C01795=1066.045,135.262,-76.737,172.704,28.495,155.211
C01796=1066.039,135.013,-76.716,172.702,28.492,155.211
C01797=1066.033,134.764,-76.696,172.701,28.489,155.210
C01798=1066.028,134.516,-76.675,172.699,28.487,155.210
C01799=1066.022,134.266,-76.654,172.697,28.484,155.209
C01800=1066.016,134.017,-76.634,172.696,28.481,155.209
C01801=1066.011,133.768,-76.613,172.694,28.478,155.209
C01802=1066.004,133.518,-76.593,172.693,28.476,155.208
C01803=1065.999,133.269,-76.572,172.691,28.473,155.208
C01804=1065.993,133.020,-76.552,172.689,28.470,155.207
C01805=1065.988,132.771,-76.532,172.687,28.467,155.207
C01806=1065.982,132.522,-76.511,172.685,28.465,155.207
C01807=1065.975,132.273,-76.490,172.684,28.462,155.206
C01808=1065.970,132.024,-76.470,172.682,28.459,155.206
C01809=1065.964,131.775,-76.450,172.680,28.456,155.205
C01810=1065.958,131.526,-76.429,172.679,28.454,155.205
C01811=1065.952,131.277,-76.409,172.677,28.451,155.205
C01812=1065.946,131.028,-76.389,172.676,28.448,155.204
C01813=1065.940,130.779,-76.369,172.674,28.445,155.204
C01814=1065.934,130.529,-76.348,172.673,28.443,155.203
C01815=1065.928,130.280,-76.328,172.671,28.440,155.203
C01816=1065.922,130.032,-76.308,172.669,28.438,155.203
C01817=1065.917,129.783,-76.288,172.667,28.435,155.202
C01818=1065.911,129.533,-76.267,172.665,28.432,155.202
C01819=1065.905,129.284,-76.247,172.664,28.429,155.201
C01820=1065.899,129.035,-76.228,172.662,28.426,155.201
C01821=1065.894,128.786,-76.208,172.660,28.424,155.201
C01822=1065.887,128.536,-76.187,172.659,28.421,155.200
C01823=1065.881,128.287,-76.167,172.657,28.418,155.200
C01824=1065.876,128.038,-76.147,172.656,28.416,155.200
C01825=1065.870,127.789,-76.127,172.654,28.413,155.199
C01826=1065.863,127.540,-76.106,172.652,28.410,155.199
C01827=1065.857,127.291,-76.086,172.651,28.408,155.198
C01828=1065.851,127.007,-76.064,172.648,28.404,155.198
C01829=1065.845,126.724,-76.041,172.647,28.401,155.197
C01830=1065.837,126.440,-76.018,172.645,28.398,155.197
C01831=1065.831,126.157,-75.995,172.643,28.395,155.197
C01832=1065.826,125.907,-75.975,172.641,28.392,155.196
C01833=1065.820,125.658,-75.955,172.640,28.390,155.196
C01834=1065.814,125.409,-75.935,172.638,28.387,155.195
C01835=1065.807,125.160,-75.915,172.636,28.384,155.195
C01836=1065.802,124.911,-75.894,172.635,28.381,155.195
C01837=1065.796,124.662,-75.874,172.633,28.379,155.194
C01838=1065.790,124.412,-75.855,172.632,28.376,155.194
C01839=1065.784,124.164,-75.835,172.630,28.373,155.193
C01840=1065.779,123.914,-75.814,172.628,28.370,155.193
C01841=1065.772,123.665,-75.794,172.627,28.368,155.193
C01842=1065.767,123.416,-75.775,172.625,28.365,155.192
C01843=1065.761,123.167,-75.755,172.624,28.363,155.192
C01844=1065.755,122.918,-75.735,172.622,28.360,155.191
C01845=1065.749,122.669,-75.714,172.620,28.357,155.191
C01846=1065.744,122.419,-75.695,172.619,28.354,155.191
C01847=1065.738,122.171,-75.675,172.617,28.352,155.190
C01848=1065.732,121.922,-75.655,172.616,28.349,155.190
C01849=1065.727,121.672,-75.635,172.614,28.346,155.189
C01850=1065.721,121.423,-75.615,172.612,28.343,155.189
C01851=1065.714,121.174,-75.595,172.610,28.340,155.189
C01852=1065.708,120.924,-75.576,172.608,28.337,155.188
C01853=1065.702,120.675,-75.556,172.607,28.335,155.188
C01854=1065.697,120.426,-75.535,172.605,28.332,155.187
C01855=1065.692,120.177,-75.516,172.604,28.329,155.187
C01856=1065.686,119.928,-75.496,172.602,28.326,155.187
C01857=1065.680,119.679,-75.476,172.601,28.324,155.186
C01858=1065.674,119.430,-75.457,172.599,28.321,155.186
C01859=1065.669,119.181,-75.436,172.597,28.318,155.185
C01860=1065.663,118.931,-75.417,172.596,28.315,155.185
C01861=1065.657,118.682,-75.397,172.594,28.313,155.185
C01862=1065.651,118.434,-75.377,172.593,28.310,155.184
C01863=1065.645,118.184,-75.358,172.591,28.307,155.184
C01864=1065.639,117.935,-75.338,172.589,28.304,155.183
C01865=1065.634,117.686,-75.318,172.588,28.302,155.183
C01866=1065.628,117.437,-75.298,172.586,28.299,155.183
C01867=1065.623,117.187,-75.279,172.585,28.296,155.182
C01868=1065.617,116.939,-75.259,172.583,28.293,155.182
C01869=1065.611,116.689,-75.240,172.582,28.291,155.181
C01870=1065.605,116.440,-75.220,172.580,28.288,155.181
C01871=1065.600,116.191,-75.200,172.578,28.285,155.181
C01872=1065.594,115.942,-75.180,172.577,28.282,155.180
C01873=1065.588,115.692,-75.161,172.575,28.280,155.180
C01874=1065.582,115.444,-75.141,172.574,28.277,155.179
C01875=1065.577,115.194,-75.122,172.572,28.274,155.179
C01876=1065.571,114.945,-75.102,172.571,28.271,155.178
C01877=1065.565,114.696,-75.082,172.569,28.268,155.178
C01878=1065.560,114.447,-75.062,172.568,28.265,155.178
C01879=1065.554,114.197,-75.043,172.566,28.262,155.177
C01880=1065.548,113.948,-75.023,172.564,28.260,155.177
C01881=1065.542,113.699,-75.003,172.563,28.257,155.176
C01882=1065.537,113.450,-74.984,172.561,28.255,155.176
C01883=1065.530,113.201,-74.965,172.560,28.252,155.176
C01884=1065.524,112.952,-74.946,172.558,28.249,155.175
C01885=1065.519,112.702,-74.926,172.556,28.246,155.175
C01886=1065.513,112.453,-74.906,172.555,28.244,155.174
C01887=1065.507,112.204,-74.887,172.553,28.241,155.174
C01888=1065.501,111.955,-74.868,172.552,28.238,155.174
C01889=1065.495,111.706,-74.848,172.550,28.235,155.173
C01890=1065.489,111.456,-74.829,172.549,28.232,155.173
C01891=1065.484,111.207,-74.809,172.547,28.230,155.172
C01892=1065.477,110.923,-74.787,172.545,28.227,155.172
C01893=1065.470,110.640,-74.765,172.543,28.223,155.172
C01894=1065.463,110.356,-74.743,172.541,28.221,155.171
C01895=1065.457,110.072,-74.721,172.540,28.217,155.171
C01896=1065.450,109.823,-74.702,172.538,28.215,155.170
C01897=1065.445,109.574,-74.683,172.537,28.212,155.170
C01898=1065.439,109.325,-74.664,172.535,28.210,155.170
C01899=1065.433,109.075,-74.644,172.534,28.207,155.169
C01900=1065.427,108.826,-74.624,172.532,28.204,155.169
C01901=1065.421,108.577,-74.606,172.530,28.201,155.168
C01902=1065.415,108.328,-74.586,172.529,28.198,155.168
C01903=1065.410,108.078,-74.567,172.527,28.196,155.168
C01904=1065.404,107.830,-74.548,172.526,28.193,155.167
C01905=1065.398,107.581,-74.529,172.524,28.190,155.167
C01906=1065.392,107.332,-74.510,172.523,28.187,155.166
C01907=1065.386,107.082,-74.490,172.521,28.185,155.166
C01908=1065.381,106.833,-74.471,172.519,28.182,155.166
C01909=1065.374,106.584,-74.453,172.518,28.180,155.165
C01910=1065.369,106.334,-74.433,172.516,28.177,155.165
C01911=1065.363,106.085,-74.414,172.515,28.174,155.164
C01912=1065.357,105.836,-74.394,172.513,28.171,155.164
C01913=1065.350,105.587,-74.375,172.512,28.169,155.164
C01914=1065.345,105.338,-74.357,172.510,28.166,155.163
C01915=1065.340,105.089,-74.337,172.508,28.163,155.163
C01916=1065.334,104.839,-74.318,172.507,28.160,155.162
C01917=1065.328,104.590,-74.299,172.505,28.157,155.162
C01918=1065.322,104.341,-74.280,172.504,28.155,155.162
C01919=1065.316,104.091,-74.261,172.502,28.152,155.161
C01920=1065.310,103.842,-74.242,172.501,28.149,155.161
C01921=1065.305,103.593,-74.223,172.499,28.146,155.160
C01922=1065.299,103.344,-74.204,172.498,28.144,155.160
C01923=1065.293,103.095,-74.185,172.497,28.141,155.160
C01924=1065.287,102.845,-74.166,172.495,28.138,155.159
C01925=1065.281,102.596,-74.147,172.494,28.136,155.159
C01926=1065.275,102.347,-74.128,172.492,28.133,155.158
C01927=1065.270,102.098,-74.110,172.491,28.130,155.158
C01928=1065.264,101.849,-74.090,172.489,28.127,155.158
C01929=1065.258,101.599,-74.071,172.488,28.124,155.157
C01930=1065.253,101.350,-74.052,172.486,28.122,155.157
C01931=1065.246,101.101,-74.033,172.484,28.119,155.156
C01932=1065.241,100.852,-74.014,172.483,28.116,155.156
C01933=1065.235,100.603,-73.996,172.481,28.114,155.156
C01934=1065.229,100.353,-73.976,172.480,28.111,155.155
C01935=1065.223,100.104,-73.958,172.478,28.108,155.155
C01936=1065.217,99.855,-73.939,172.477,28.106,155.154
C01937=1065.210,99.606,-73.920,172.475,28.103,155.154
C01938=1065.205,99.356,-73.901,172.473,28.100,155.154
C01939=1065.199,99.108,-73.882,172.472,28.097,155.153
C01940=1065.193,98.859,-73.863,172.470,28.094,155.153
C01941=1065.187,98.609,-73.845,172.469,28.092,155.153
C01942=1065.181,98.359,-73.826,172.467,28.089,155.152
C01943=1065.175,98.110,-73.807,172.466,28.087,155.152
C01944=1065.170,97.862,-73.788,172.464,28.084,155.151
C01945=1065.163,97.612,-73.770,172.462,28.081,155.151
C01946=1065.158,97.363,-73.751,172.461,28.078,155.151
C01947=1065.151,97.114,-73.732,172.460,28.076,155.150
C01948=1065.146,96.864,-73.713,172.459,28.073,155.150
C01949=1065.140,96.615,-73.695,172.457,28.070,155.149
C01950=1065.134,96.366,-73.676,172.456,28.067,155.149
C01951=1065.128,96.117,-73.657,172.454,28.065,155.149
C01952=1065.122,95.867,-73.639,172.452,28.062,155.148
C01953=1065.117,95.618,-73.620,172.451,28.060,155.148
C01954=1065.110,95.369,-73.602,172.449,28.057,155.147
C01955=1065.105,95.120,-73.582,172.448,28.054,155.147
C01956=1065.098,94.836,-73.561,172.446,28.051,155.147
C01957=1065.091,94.553,-73.541,172.445,28.048,155.146
C01958=1065.085,94.268,-73.519,172.442,28.044,155.146
C01959=1065.078,93.985,-73.497,172.441,28.042,155.145
C01960=1065.072,93.736,-73.480,172.439,28.039,155.145
C01961=1065.067,93.486,-73.461,172.438,28.036,155.144
C01962=1065.060,93.237,-73.442,172.436,28.033,155.144
C01963=1065.055,92.988,-73.424,172.435,28.030,155.144
C01964=1065.049,92.739,-73.405,172.433,28.028,155.143
C01965=1065.043,92.490,-73.387,172.431,28.025,155.143
C01966=1065.037,92.240,-73.368,172.431,28.022,155.142
C01967=1065.031,91.991,-73.350,172.429,28.020,155.142
C01968=1065.026,91.742,-73.330,172.428,28.017,155.142
C01969=1065.020,91.492,-73.313,172.426,28.014,155.141
C01970=1065.014,91.244,-73.294,172.425,28.011,155.141
C01971=1065.008,90.994,-73.275,172.423,28.009,155.141
C01972=1065.002,90.745,-73.257,172.421,28.006,155.140
C01973=1064.996,90.496,-73.239,172.420,28.003,155.140
C01974=1064.991,90.246,-73.220,172.418,28.001,155.139
C01975=1064.984,89.997,-73.202,172.417,27.998,155.139
C01976=1064.979,89.748,-73.184,172.415,27.995,155.139
C01977=1064.972,89.499,-73.165,172.414,27.992,155.138
C01978=1064.966,89.250,-73.147,172.412,27.990,155.138
C01979=1064.961,89.000,-73.128,172.410,27.987,155.137
C01980=1064.955,88.751,-73.110,172.409,27.985,155.137
C01981=1064.949,88.501,-73.092,172.408,27.982,155.137
C01982=1064.942,88.252,-73.073,172.407,27.979,155.136
C01983=1064.937,88.003,-73.056,172.405,27.976,155.136
C01984=1064.931,87.754,-73.037,172.404,27.974,155.135
C01985=1064.925,87.504,-73.019,172.402,27.971,155.135
C01986=1064.919,87.256,-73.000,172.401,27.969,155.135
C01987=1064.913,87.006,-72.982,172.399,27.966,155.134
C01988=1064.906,86.757,-72.964,172.397,27.963,155.134
C01989=1064.901,86.508,-72.946,172.396,27.960,155.134
C01990=1064.896,86.258,-72.928,172.394,27.957,155.133
C01991=1064.889,86.009,-72.909,172.393,27.955,155.133
C01992=1064.884,85.760,-72.891,172.391,27.952,155.132
C01993=1064.877,85.510,-72.873,172.390,27.949,155.132
C01994=1064.871,85.261,-72.855,172.388,27.947,155.132
C01995=1064.865,85.012,-72.837,172.387,27.944,155.131
C01996=1064.859,84.763,-72.819,172.386,27.942,155.131
C01997=1064.854,84.513,-72.800,172.384,27.939,155.130
C01998=1064.848,84.264,-72.782,172.383,27.936,155.130
C01999=1064.842,84.014,-72.764,172.381,27.933,155.130
C02000=1064.836,83.766,-72.746,172.380,27.930,155.129
C02001=1064.830,83.516,-72.728,172.378,27.928,155.129
C02002=1064.824,83.267,-72.710,172.377,27.925,155.128
C02003=1064.818,83.018,-72.691,172.375,27.922,155.128
C02004=1064.812,82.768,-72.674,172.373,27.920,155.128
C02005=1064.807,82.519,-72.655,172.372,27.917,155.127
C02006=1064.801,82.270,-72.637,172.370,27.914,155.127
C02007=1064.795,82.021,-72.619,172.370,27.912,155.127
C02008=1064.789,81.771,-72.601,172.368,27.909,155.126
C02009=1064.783,81.522,-72.584,172.367,27.906,155.126
C02010=1064.777,81.273,-72.565,172.365,27.903,155.125
C02011=1064.771,81.024,-72.547,172.364,27.900,155.125
C02012=1064.765,80.774,-72.530,172.362,27.898,155.125
C02013=1064.760,80.526,-72.511,172.361,27.895,155.124
C02014=1064.754,80.276,-72.493,172.359,27.892,155.124
C02015=1064.748,80.026,-72.475,172.357,27.889,155.123
C02016=1064.743,79.777,-72.457,172.356,27.887,155.123
C02017=1064.736,79.528,-72.439,172.354,27.884,155.123
C02018=1064.731,79.279,-72.421,172.354,27.882,155.122
C02019=1064.724,79.029,-72.403,172.352,27.879,155.122
C02020=1064.718,78.746,-72.382,172.350,27.875,155.121
C02021=1064.711,78.462,-72.363,172.348,27.873,155.121
C02022=1064.704,78.178,-72.342,172.347,27.869,155.120
C02023=1064.698,77.894,-72.322,172.345,27.866,155.120
C02024=1064.692,77.645,-72.303,172.344,27.864,155.120
C02025=1064.686,77.396,-72.286,172.342,27.861,155.119
C02026=1064.680,77.146,-72.268,172.341,27.858,155.119
C02027=1064.674,76.898,-72.251,172.339,27.855,155.118
C02028=1064.668,76.648,-72.233,172.338,27.853,155.118
C02029=1064.662,76.399,-72.216,172.336,27.850,155.118
C02030=1064.656,76.149,-72.198,172.335,27.848,155.117
C02031=1064.650,75.901,-72.179,172.334,27.845,155.117
C02032=1064.644,75.651,-72.161,172.332,27.842,155.117
C02033=1064.639,75.402,-72.144,172.331,27.839,155.116
C02034=1064.633,75.152,-72.126,172.329,27.836,155.116
C02035=1064.626,74.903,-72.109,172.328,27.834,155.115
C02036=1064.620,74.654,-72.091,172.326,27.831,155.115
C02037=1064.615,74.405,-72.073,172.325,27.829,155.115
C02038=1064.609,74.155,-72.055,172.323,27.826,155.114
C02039=1064.603,73.906,-72.038,172.321,27.823,155.114
C02040=1064.597,73.656,-72.020,172.321,27.820,155.113
C02041=1064.591,73.407,-72.002,172.319,27.818,155.113
C02042=1064.585,73.158,-71.985,172.318,27.815,155.113
C02043=1064.579,72.909,-71.967,172.316,27.813,155.112
C02044=1064.573,72.659,-71.950,172.315,27.810,155.112
C02045=1064.567,72.410,-71.932,172.313,27.807,155.112
C02046=1064.561,72.160,-71.914,172.312,27.804,155.111
C02047=1064.556,71.911,-71.896,172.310,27.801,155.111
C02048=1064.549,71.662,-71.880,172.309,27.799,155.110
C02049=1064.543,71.413,-71.862,172.307,27.796,155.110
C02050=1064.538,71.164,-71.844,172.305,27.794,155.110
C02051=1064.532,70.914,-71.826,172.305,27.791,155.109
C02052=1064.526,70.665,-71.809,172.303,27.788,155.109
C02053=1064.519,70.415,-71.791,172.302,27.785,155.108
C02054=1064.514,70.166,-71.774,172.300,27.783,155.108
C02055=1064.508,69.917,-71.756,172.299,27.780,155.108
C02056=1064.502,69.667,-71.739,172.297,27.777,155.107
C02057=1064.496,69.418,-71.722,172.296,27.774,155.107
C02058=1064.490,69.168,-71.704,172.294,27.772,155.107
C02059=1064.485,68.919,-71.686,172.292,27.769,155.106
C02060=1064.478,68.670,-71.669,172.292,27.767,155.106
C02061=1064.472,68.421,-71.651,172.290,27.764,155.105
C02062=1064.467,68.172,-71.634,172.289,27.761,155.105
C02063=1064.460,67.922,-71.617,172.287,27.758,155.105
C02064=1064.455,67.673,-71.600,172.286,27.756,155.104
C02065=1064.449,67.423,-71.582,172.284,27.753,155.104
C02066=1064.442,67.174,-71.565,172.283,27.750,155.104
C02067=1064.437,66.925,-71.547,172.281,27.748,155.103
C02068=1064.431,66.676,-71.529,172.280,27.745,155.103
C02069=1064.425,66.426,-71.513,172.278,27.742,155.102
C02070=1064.419,66.176,-71.495,172.277,27.740,155.102
C02071=1064.413,65.927,-71.478,172.276,27.737,155.102
C02072=1064.407,65.679,-71.461,172.274,27.734,155.101
C02073=1064.401,65.428,-71.443,172.273,27.732,155.101
C02074=1064.395,65.180,-71.426,172.271,27.729,155.100
C02075=1064.389,64.931,-71.409,172.270,27.726,155.100
C02076=1064.383,64.681,-71.391,172.268,27.723,155.100
C02077=1064.377,64.431,-71.375,172.267,27.721,155.099
C02078=1064.371,64.182,-71.357,172.265,27.718,155.099
C02079=1064.365,63.933,-71.340,172.265,27.716,155.099
C02080=1064.360,63.683,-71.323,172.263,27.713,155.098
C02081=1064.353,63.434,-71.306,172.261,27.711,155.098
C02082=1064.346,63.185,-71.289,172.260,27.708,155.097
C02083=1064.340,62.935,-71.271,172.258,27.705,155.097
C02084=1064.334,62.651,-71.252,172.257,27.702,155.097
C02085=1064.327,62.368,-71.233,172.255,27.699,155.096
C02086=1064.320,62.084,-71.213,172.253,27.696,155.096
C02087=1064.313,61.800,-71.194,172.251,27.693,155.095
C02088=1064.306,61.551,-71.177,172.250,27.691,155.095
C02089=1064.301,61.302,-71.159,172.248,27.688,155.095
C02090=1064.294,61.052,-71.142,172.248,27.685,155.094
C02091=1064.289,60.803,-71.125,172.246,27.682,155.094
C02092=1064.282,60.553,-71.108,172.245,27.680,155.094
C02093=1064.276,60.304,-71.091,172.243,27.677,155.093
C02094=1064.271,60.055,-71.074,172.242,27.675,155.093
C02095=1064.264,59.805,-71.057,172.240,27.672,155.092
C02096=1064.258,59.556,-71.040,172.238,27.670,155.092
C02097=1064.253,59.307,-71.023,172.237,27.667,155.092
C02098=1064.246,59.057,-71.006,172.235,27.664,155.091
C02099=1064.240,58.808,-70.990,172.235,27.661,155.091
C02100=1064.234,58.559,-70.972,172.233,27.659,155.091
C02101=1064.228,58.310,-70.956,172.232,27.656,155.090
C02102=1064.222,58.060,-70.938,172.230,27.653,155.090
C02103=1064.216,57.810,-70.922,172.229,27.651,155.089
C02104=1064.210,57.562,-70.905,172.227,27.648,155.089
C02105=1064.204,57.311,-70.887,172.225,27.646,155.089
C02106=1064.198,57.063,-70.871,172.224,27.643,155.088
C02107=1064.192,56.813,-70.854,172.222,27.640,155.088
C02108=1064.186,56.564,-70.837,172.222,27.637,155.088
C02109=1064.180,56.314,-70.820,172.220,27.635,155.087
C02110=1064.174,56.065,-70.803,172.219,27.632,155.087
C02111=1064.168,55.816,-70.786,172.217,27.630,155.087
C02112=1064.162,55.566,-70.769,172.216,27.627,155.086
C02113=1064.156,55.317,-70.753,172.214,27.624,155.086
C02114=1064.150,55.068,-70.736,172.213,27.622,155.085
C02115=1064.144,54.819,-70.719,172.211,27.619,155.085
C02116=1064.138,54.569,-70.703,172.210,27.616,155.085
C02117=1064.131,54.320,-70.685,172.209,27.613,155.084
C02118=1064.126,54.070,-70.668,172.207,27.611,155.084
C02119=1064.120,53.821,-70.652,172.206,27.608,155.084
C02120=1064.114,53.572,-70.635,172.204,27.606,155.083
C02121=1064.108,53.322,-70.618,172.203,27.603,155.083
C02122=1064.102,53.072,-70.602,172.201,27.601,155.082
C02123=1064.096,52.824,-70.585,172.200,27.598,155.082
C02124=1064.091,52.574,-70.568,172.198,27.595,155.082
C02125=1064.085,52.325,-70.552,172.197,27.592,155.081
C02126=1064.078,52.075,-70.534,172.196,27.590,155.081
C02127=1064.072,51.826,-70.518,172.195,27.587,155.081
C02128=1064.067,51.576,-70.501,172.193,27.584,155.080
C02129=1064.060,51.327,-70.484,172.192,27.582,155.080
C02130=1064.054,51.078,-70.468,172.190,27.579,155.079
C02131=1064.049,50.828,-70.451,172.188,27.576,155.079
C02132=1064.042,50.579,-70.434,172.187,27.574,155.079
C02133=1064.036,50.330,-70.417,172.185,27.571,155.078
C02134=1064.030,50.080,-70.401,172.185,27.568,155.078
C02135=1064.025,49.831,-70.384,172.183,27.566,155.078
C02136=1064.019,49.582,-70.367,172.182,27.563,155.077
C02137=1064.013,49.333,-70.351,172.180,27.560,155.077
C02138=1064.007,49.083,-70.335,172.179,27.558,155.076
C02139=1064.001,48.833,-70.318,172.177,27.555,155.076
C02140=1063.995,48.584,-70.301,172.176,27.552,155.076
C02141=1063.989,48.335,-70.284,172.174,27.549,155.075
C02142=1063.983,48.085,-70.268,172.173,27.546,155.075
C02143=1063.978,47.836,-70.251,172.172,27.544,155.075
C02144=1063.972,47.586,-70.235,172.170,27.542,155.074
C02145=1063.966,47.337,-70.219,172.169,27.539,155.074
C02146=1063.960,47.088,-70.202,172.167,27.536,155.073
C02147=1063.955,46.839,-70.185,172.166,27.533,155.073
C02148=1063.948,46.555,-70.166,172.164,27.530,155.073
C02149=1063.940,46.270,-70.148,172.163,27.527,155.072
C02150=1063.933,45.986,-70.129,172.162,27.524,155.072
C02151=1063.927,45.702,-70.110,172.160,27.521,155.071
C02152=1063.922,45.453,-70.093,172.159,27.518,155.071
C02153=1063.916,45.203,-70.077,172.157,27.516,155.070
C02154=1063.910,44.954,-70.061,172.156,27.513,155.070
C02155=1063.904,44.704,-70.044,172.154,27.510,155.070
C02156=1063.898,44.455,-70.028,172.152,27.508,155.069
C02157=1063.893,44.205,-70.011,172.151,27.505,155.069
C02158=1063.886,43.957,-69.994,172.149,27.502,155.069
C02159=1063.880,43.707,-69.978,172.148,27.499,155.068
C02160=1063.874,43.458,-69.962,172.147,27.497,155.068
C02161=1063.869,43.209,-69.946,172.146,27.494,155.068
C02162=1063.863,42.959,-69.929,172.144,27.492,155.067
C02163=1063.856,42.709,-69.913,172.143,27.489,155.067
C02164=1063.850,42.460,-69.896,172.141,27.486,155.066
C02165=1063.844,42.211,-69.880,172.140,27.484,155.066
C02166=1063.838,41.961,-69.864,172.138,27.481,155.066
C02167=1063.832,41.712,-69.848,172.137,27.478,155.065
C02168=1063.826,41.463,-69.831,172.136,27.476,155.065
C02169=1063.820,41.213,-69.815,172.134,27.473,155.065
C02170=1063.814,40.964,-69.799,172.133,27.470,155.064
C02171=1063.808,40.715,-69.783,172.131,27.468,155.064
C02172=1063.802,40.465,-69.766,172.130,27.465,155.064
C02173=1063.797,40.215,-69.751,172.128,27.462,155.063
C02174=1063.791,39.966,-69.735,172.127,27.460,155.063
C02175=1063.785,39.717,-69.718,172.125,27.457,155.062
C02176=1063.779,39.467,-69.702,172.124,27.455,155.062
C02177=1063.773,39.218,-69.686,172.123,27.452,155.062
C02178=1063.767,38.968,-69.670,172.122,27.449,155.061
C02179=1063.761,38.719,-69.653,172.120,27.447,155.061
C02180=1063.755,38.470,-69.637,172.119,27.444,155.061
C02181=1063.749,38.220,-69.621,172.117,27.441,155.060
C02182=1063.743,37.971,-69.605,172.116,27.438,155.060
C02183=1063.738,37.721,-69.589,172.114,27.436,155.060
C02184=1063.731,37.472,-69.573,172.113,27.433,155.059
C02185=1063.725,37.223,-69.557,172.111,27.431,155.059
C02186=1063.719,36.973,-69.541,172.110,27.429,155.058
C02187=1063.713,36.724,-69.525,172.109,27.426,155.058
C02188=1063.707,36.475,-69.508,172.107,27.423,155.058
C02189=1063.701,36.225,-69.493,172.106,27.421,155.057
C02190=1063.695,35.976,-69.477,172.104,27.418,155.057
C02191=1063.689,35.726,-69.461,172.103,27.416,155.057
C02192=1063.683,35.477,-69.445,172.101,27.413,155.056
C02193=1063.677,35.228,-69.428,172.100,27.410,155.056
C02194=1063.671,34.978,-69.413,172.098,27.408,155.056
C02195=1063.665,34.729,-69.397,172.098,27.405,155.055
C02196=1063.659,34.479,-69.381,172.096,27.402,155.055
C02197=1063.653,34.230,-69.365,172.094,27.400,155.055
C02198=1063.646,33.980,-69.350,172.093,27.397,155.054
C02199=1063.640,33.731,-69.333,172.091,27.394,155.054
C02200=1063.634,33.482,-69.317,172.090,27.392,155.053
C02201=1063.629,33.232,-69.302,172.088,27.389,155.053
C02202=1063.622,32.983,-69.286,172.087,27.386,155.053
C02203=1063.616,32.733,-69.270,172.086,27.384,155.052
C02204=1063.610,32.484,-69.253,172.085,27.382,155.052
C02205=1063.605,32.234,-69.238,172.083,27.379,155.052
C02206=1063.598,31.985,-69.222,172.082,27.376,155.051
C02207=1063.592,31.736,-69.206,172.080,27.374,155.051
C02208=1063.586,31.486,-69.190,172.079,27.371,155.051
C02209=1063.580,31.236,-69.174,172.077,27.368,155.050
C02210=1063.574,30.987,-69.158,172.076,27.366,155.050
C02211=1063.569,30.738,-69.143,172.074,27.363,155.050
C02212=1063.561,30.454,-69.125,172.073,27.360,155.049
C02213=1063.555,30.170,-69.107,172.071,27.357,155.049
C02214=1063.548,29.885,-69.089,172.070,27.354,155.048
C02215=1063.541,29.601,-69.071,172.068,27.351,155.048
C02216=1063.535,29.352,-69.055,172.067,27.349,155.048
C02217=1063.529,29.102,-69.040,172.065,27.346,155.047
C02218=1063.523,28.853,-69.023,172.064,27.344,155.047
C02219=1063.517,28.603,-69.008,172.062,27.341,155.046
C02220=1063.511,28.354,-68.992,172.061,27.338,155.046
C02221=1063.506,28.105,-68.977,172.059,27.336,155.046
C02222=1063.499,27.855,-68.961,172.058,27.334,155.046
C02223=1063.493,27.605,-68.946,172.057,27.331,155.045
C02224=1063.487,27.356,-68.930,172.055,27.328,155.045
C02225=1063.481,27.106,-68.914,172.054,27.326,155.044
C02226=1063.474,26.857,-68.899,172.052,27.323,155.044
C02227=1063.469,26.607,-68.883,172.051,27.321,155.044
C02228=1063.463,26.358,-68.867,172.049,27.318,155.043
C02229=1063.456,26.108,-68.852,172.048,27.315,155.043
C02230=1063.451,25.860,-68.836,172.046,27.313,155.043
C02231=1063.445,25.610,-68.821,172.046,27.310,155.042
C02232=1063.439,25.361,-68.805,172.044,27.308,155.042
C02233=1063.432,25.111,-68.790,172.043,27.305,155.042
C02234=1063.426,24.862,-68.774,172.041,27.303,155.041
C02235=1063.420,24.612,-68.759,172.039,27.300,155.041
C02236=1063.414,24.363,-68.743,172.038,27.298,155.041
C02237=1063.408,24.114,-68.728,172.036,27.295,155.040
C02238=1063.403,23.864,-68.712,172.035,27.292,155.040
C02239=1063.396,23.615,-68.697,172.033,27.290,155.040
C02240=1063.390,23.365,-68.681,172.032,27.287,155.039
C02241=1063.384,23.116,-68.666,172.031,27.285,155.039
C02242=1063.378,22.866,-68.650,172.030,27.282,155.039
C02243=1063.372,22.617,-68.635,172.028,27.280,155.038
C02244=1063.366,22.368,-68.619,172.027,27.277,155.038
C02245=1063.360,22.118,-68.604,172.025,27.274,155.037
C02246=1063.354,21.868,-68.589,172.024,27.272,155.037
C02247=1063.347,21.619,-68.573,172.022,27.269,155.037
C02248=1063.342,21.370,-68.558,172.021,27.267,155.037
C02249=1063.336,21.120,-68.543,172.019,27.264,155.036
C02250=1063.330,20.871,-68.527,172.018,27.262,155.036
C02251=1063.324,20.621,-68.512,172.017,27.259,155.035
C02252=1063.318,20.371,-68.496,172.015,27.257,155.035
C02253=1063.312,20.123,-68.481,172.014,27.254,155.035
C02254=1063.306,19.873,-68.466,172.012,27.252,155.035
C02255=1063.300,19.623,-68.450,172.011,27.249,155.034
C02256=1063.293,19.374,-68.435,172.009,27.246,155.034
C02257=1063.287,19.124,-68.420,172.008,27.244,155.033
C02258=1063.282,18.875,-68.405,172.006,27.241,155.033
C02259=1063.275,18.625,-68.390,172.005,27.238,155.033
C02260=1063.270,18.376,-68.373,172.004,27.236,155.033
C02261=1063.263,18.126,-68.358,172.003,27.234,155.032
C02262=1063.257,17.877,-68.344,172.001,27.231,155.032
C02263=1063.252,17.628,-68.328,171.999,27.229,155.031
C02264=1063.245,17.378,-68.313,171.998,27.226,155.031
C02265=1063.239,17.129,-68.298,171.996,27.223,155.031
C02266=1063.234,16.880,-68.283,171.995,27.221,155.031
C02267=1063.227,16.630,-68.268,171.993,27.218,155.030
C02268=1063.221,16.380,-68.253,171.992,27.216,155.030
C02269=1063.215,16.130,-68.237,171.990,27.213,155.029
C02270=1063.209,15.881,-68.223,171.990,27.211,155.029
C02271=1063.203,15.632,-68.207,171.988,27.208,155.029
C02272=1063.197,15.382,-68.191,171.987,27.206,155.028
C02273=1063.191,15.133,-68.176,171.985,27.203,155.028
C02274=1063.185,14.884,-68.162,171.984,27.201,155.028
C02275=1063.179,14.634,-68.146,171.982,27.198,155.027
C02276=1063.172,14.351,-68.129,171.981,27.195,155.027
C02277=1063.165,14.069,-68.113,171.979,27.192,155.027
C02278=1063.158,13.786,-68.095,171.978,27.190,155.026
C02279=1063.151,13.503,-68.078,171.975,27.187,155.026
C02280=1063.145,13.254,-68.063,171.974,27.184,155.026
C02281=1063.139,13.004,-68.048,171.973,27.182,155.025
C02282=1063.132,12.754,-68.033,171.972,27.179,155.025
C02283=1063.126,12.505,-68.018,171.970,27.177,155.025
C02284=1063.120,12.256,-68.004,171.968,27.175,155.024
C02285=1063.114,12.006,-67.989,171.967,27.172,155.024
C02286=1063.108,11.757,-67.974,171.965,27.170,155.024
C02287=1063.103,11.507,-67.959,171.964,27.167,155.023
C02288=1063.096,11.258,-67.944,171.962,27.165,155.023
C02289=1063.090,11.008,-67.929,171.961,27.162,155.023
C02290=1063.083,10.758,-67.914,171.959,27.159,155.022
C02291=1063.078,10.509,-67.899,171.958,27.157,155.022
C02292=1063.071,10.260,-67.884,171.956,27.155,155.022
C02293=1063.065,10.010,-67.869,171.956,27.152,155.021
C02294=1063.059,9.761,-67.855,171.954,27.150,155.021
C02295=1063.053,9.511,-67.840,171.952,27.148,155.021
C02296=1063.046,9.262,-67.825,171.951,27.145,155.021
C02297=1063.040,9.013,-67.810,171.949,27.143,155.020
C02298=1063.035,8.763,-67.795,171.948,27.140,155.020
C02299=1063.028,8.513,-67.780,171.946,27.137,155.020
C02300=1063.023,8.264,-67.766,171.945,27.135,155.019
C02301=1063.017,8.014,-67.751,171.943,27.132,155.019
C02302=1063.010,7.764,-67.736,171.942,27.130,155.019
C02303=1063.004,7.515,-67.722,171.940,27.128,155.018
C02304=1062.998,7.266,-67.707,171.940,27.125,155.018
C02305=1062.992,7.017,-67.692,171.938,27.123,155.018
C02306=1062.986,6.767,-67.677,171.936,27.121,155.017
C02307=1062.980,6.517,-67.662,171.935,27.118,155.017
C02308=1062.974,6.268,-67.648,171.933,27.115,155.017
C02309=1062.968,6.018,-67.633,171.932,27.113,155.017
C02310=1062.961,5.769,-67.618,171.930,27.110,155.016
C02311=1062.955,5.520,-67.604,171.929,27.108,155.016
C02312=1062.949,5.270,-67.589,171.927,27.105,155.015
C02313=1062.943,5.021,-67.574,171.926,27.103,155.015
C02314=1062.937,4.771,-67.560,171.924,27.101,155.015
C02315=1062.931,4.522,-67.545,171.923,27.098,155.015
C02316=1062.925,4.272,-67.531,171.921,27.096,155.014
C02317=1062.919,4.022,-67.515,171.920,27.094,155.014
C02318=1062.914,3.773,-67.500,171.919,27.091,155.014
C02319=1062.908,3.523,-67.486,171.917,27.088,155.013
C02320=1062.902,3.274,-67.472,171.916,27.086,155.013
C02321=1062.895,3.024,-67.457,171.914,27.083,155.013
C02322=1062.890,2.775,-67.442,171.913,27.081,155.012
C02323=1062.884,2.525,-67.428,171.911,27.079,155.012
C02324=1062.877,2.275,-67.413,171.910,27.076,155.012
C02325=1062.871,2.026,-67.398,171.908,27.074,155.011
C02326=1062.865,1.777,-67.383,171.907,27.071,155.011
C02327=1062.860,1.527,-67.370,171.905,27.068,155.011
C02328=1062.853,1.278,-67.355,171.904,27.066,155.011
C02329=1062.847,1.029,-67.340,171.903,27.064,155.010
C02330=1062.841,0.778,-67.326,171.902,27.061,155.010
C02331=1062.835,0.529,-67.311,171.900,27.059,155.010
C02332=1062.829,0.280,-67.296,171.899,27.056,155.009
C02333=1062.824,0.030,-67.282,171.897,27.054,155.009
C02334=1062.817,-0.220,-67.267,171.895,27.052,155.009
C02335=1062.811,-0.469,-67.253,171.894,27.049,155.008
C02336=1062.805,-0.719,-67.239,171.892,27.046,155.008
C02337=1062.800,-0.968,-67.224,171.891,27.044,155.008
C02338=1062.793,-1.217,-67.209,171.889,27.041,155.007
C02339=1062.787,-1.467,-67.196,171.888,27.039,155.007
C02340=1062.781,-1.747,-67.179,171.886,27.036,155.007
C02341=1062.774,-2.029,-67.163,171.885,27.034,155.006
C02342=1062.767,-2.309,-67.146,171.883,27.031,155.006
C02343=1062.761,-2.590,-67.131,171.882,27.028,155.006
C02344=1062.754,-2.839,-67.116,171.880,27.026,155.005
C02345=1062.749,-3.089,-67.102,171.879,27.023,155.005
C02346=1062.743,-3.339,-67.087,171.877,27.021,155.005
C02347=1062.737,-3.588,-67.073,171.876,27.018,155.004
C02348=1062.730,-3.838,-67.059,171.874,27.016,155.004
C02349=1062.724,-4.087,-67.045,171.872,27.014,155.004
C02350=1062.718,-4.337,-67.030,171.871,27.011,155.003
C02351=1062.712,-4.586,-67.017,171.869,27.009,155.003
C02352=1062.705,-4.836,-67.002,171.868,27.006,155.003
C02353=1062.700,-5.085,-66.988,171.866,27.004,155.003
C02354=1062.693,-5.335,-66.973,171.865,27.002,155.002
C02355=1062.687,-5.584,-66.960,171.863,27.000,155.002
C02356=1062.681,-5.834,-66.945,171.862,26.997,155.002
C02357=1062.676,-6.083,-66.931,171.860,26.994,155.001
C02358=1062.668,-6.333,-66.916,171.860,26.992,155.001
C02359=1062.663,-6.582,-66.902,171.858,26.990,155.001
C02360=1062.657,-6.833,-66.888,171.856,26.988,155.001
C02361=1062.650,-7.081,-66.874,171.855,26.986,155.000
C02362=1062.645,-7.331,-66.860,171.853,26.983,155.000
C02363=1062.638,-7.581,-66.845,171.852,26.980,155.000
C02364=1062.632,-7.830,-66.832,171.850,26.978,154.999
C02365=1062.626,-8.079,-66.817,171.849,26.976,154.999
C02366=1062.620,-8.329,-66.803,171.847,26.974,154.999
C02367=1062.614,-8.579,-66.790,171.846,26.971,154.999
C02368=1062.608,-8.828,-66.775,171.844,26.969,154.998
C02369=1062.602,-9.078,-66.761,171.842,26.967,154.998
C02370=1062.596,-9.327,-66.748,171.841,26.964,154.998
C02371=1062.590,-9.576,-66.733,171.839,26.962,154.997
C02372=1062.584,-9.827,-66.719,171.838,26.959,154.997
C02373=1062.577,-10.076,-66.706,171.836,26.957,154.997
C02374=1062.572,-10.325,-66.691,171.835,26.955,154.997
C02375=1062.565,-10.575,-66.677,171.833,26.952,154.996
C02376=1062.559,-10.824,-66.664,171.832,26.950,154.996
C02377=1062.553,-11.074,-66.649,171.831,26.947,154.996
C02378=1062.547,-11.323,-66.635,171.830,26.945,154.995
C02379=1062.541,-11.573,-66.621,171.828,26.943,154.995
C02380=1062.535,-11.823,-66.606,171.826,26.941,154.995
C02381=1062.529,-12.072,-66.593,171.825,26.938,154.995
C02382=1062.523,-12.321,-66.579,171.823,26.936,154.994
C02383=1062.517,-12.572,-66.565,171.822,26.934,154.994
C02384=1062.511,-12.820,-66.551,171.820,26.931,154.994
C02385=1062.505,-13.070,-66.537,171.819,26.929,154.993
C02386=1062.498,-13.320,-66.524,171.817,26.926,154.993
C02387=1062.493,-13.570,-66.510,171.816,26.924,154.993
C02388=1062.487,-13.819,-66.496,171.814,26.922,154.993
C02389=1062.480,-14.068,-66.482,171.813,26.919,154.992
C02390=1062.475,-14.318,-66.468,171.811,26.917,154.992
C02391=1062.469,-14.567,-66.454,171.809,26.915,154.992
C02392=1062.463,-14.818,-66.440,171.808,26.913,154.992
C02393=1062.457,-15.067,-66.426,171.806,26.910,154.991
C02394=1062.451,-15.316,-66.412,171.805,26.908,154.991
C02395=1062.444,-15.566,-66.399,171.803,26.906,154.991
C02396=1062.438,-15.815,-66.385,171.802,26.903,154.990
C02397=1062.432,-16.065,-66.372,171.800,26.901,154.990
C02398=1062.426,-16.315,-66.357,171.799,26.899,154.990
C02399=1062.420,-16.564,-66.344,171.798,26.897,154.990
C02400=1062.414,-16.814,-66.330,171.796,26.894,154.989
C02401=1062.407,-17.064,-66.317,171.795,26.892,154.989
C02402=1062.401,-17.312,-66.303,171.793,26.890,154.989
C02403=1062.395,-17.562,-66.289,171.792,26.888,154.989
C02404=1062.386,-17.913,-66.270,171.789,26.884,154.988
C02405=1062.378,-18.262,-66.251,171.787,26.881,154.988
C02406=1062.369,-18.612,-66.232,171.785,26.878,154.987
C02407=1062.361,-18.962,-66.212,171.783,26.875,154.987
C02408=1062.355,-19.211,-66.199,171.782,26.872,154.987
C02409=1062.349,-19.461,-66.185,171.780,26.870,154.987
C02410=1062.342,-19.710,-66.171,171.778,26.868,154.986
C02411=1062.336,-19.960,-66.158,171.777,26.866,154.986
C02412=1062.330,-20.210,-66.144,171.775,26.864,154.986
C02413=1062.324,-20.459,-66.131,171.774,26.862,154.986
C02414=1062.318,-20.709,-66.117,171.772,26.859,154.985
C02415=1062.312,-20.958,-66.104,171.771,26.857,154.985
C02416=1062.305,-21.208,-66.090,171.769,26.855,154.985
C02417=1062.299,-21.457,-66.077,171.767,26.852,154.985
C02418=1062.294,-21.707,-66.063,171.766,26.850,154.984
C02419=1062.288,-21.956,-66.050,171.764,26.848,154.984
C02420=1062.281,-22.206,-66.035,171.763,26.845,154.984
C02421=1062.275,-22.456,-66.022,171.761,26.843,154.983
C02422=1062.269,-22.705,-66.009,171.760,26.841,154.983
C02423=1062.264,-22.955,-65.996,171.758,26.839,154.983
C02424=1062.258,-23.204,-65.982,171.757,26.836,154.983
C02425=1062.251,-23.454,-65.969,171.755,26.834,154.982
C02426=1062.245,-23.704,-65.955,171.753,26.832,154.982
C02427=1062.239,-23.953,-65.942,171.752,26.830,154.982
C02428=1062.233,-24.202,-65.928,171.750,26.828,154.982
C02429=1062.227,-24.452,-65.914,171.749,26.825,154.981
C02430=1062.221,-24.701,-65.901,171.747,26.823,154.981
C02431=1062.214,-24.951,-65.888,171.746,26.821,154.981
C02432=1062.210,-25.165,-65.876,171.745,26.819,154.981
C02433=1062.204,-25.380,-65.865,171.743,26.817,154.980
C02434=1062.199,-25.594,-65.853,171.742,26.815,154.980
C02435=1062.194,-25.809,-65.842,171.741,26.813,154.980
C02436=1062.188,-26.022,-65.830,171.739,26.812,154.980
C02437=1062.184,-26.236,-65.819,171.738,26.809,154.980
C02438=1062.179,-26.451,-65.808,171.736,26.808,154.979
C02439=1062.173,-26.665,-65.796,171.736,26.806,154.979
C02440=1062.168,-26.914,-65.782,171.734,26.803,154.979
C02441=1062.162,-27.164,-65.769,171.732,26.801,154.979
C02442=1062.156,-27.414,-65.756,171.731,26.799,154.978
C02443=1062.149,-27.664,-65.743,171.729,26.797,154.978
C02444=1062.142,-27.913,-65.729,171.728,26.795,154.978
C02445=1062.137,-28.163,-65.717,171.726,26.792,154.978
C02446=1062.130,-28.412,-65.703,171.725,26.791,154.977
C02447=1062.124,-28.661,-65.690,171.723,26.788,154.977
C02448=1062.117,-28.911,-65.677,171.721,26.786,154.977
C02449=1062.112,-29.161,-65.663,171.720,26.784,154.977
C02450=1062.106,-29.411,-65.650,171.718,26.782,154.977
C02451=1062.100,-29.660,-65.637,171.717,26.780,154.976
C02452=1062.094,-29.909,-65.624,171.715,26.777,154.976
C02453=1062.088,-30.159,-65.611,171.713,26.776,154.976
C02454=1062.081,-30.408,-65.598,171.712,26.773,154.976
C02455=1062.075,-30.658,-65.584,171.710,26.771,154.975
C02456=1062.069,-30.908,-65.572,171.709,26.769,154.975
C02457=1062.062,-31.157,-65.558,171.707,26.767,154.975
C02458=1062.056,-31.407,-65.545,171.706,26.765,154.975
C02459=1062.050,-31.657,-65.533,171.704,26.762,154.974
C02460=1062.044,-31.906,-65.519,171.702,26.761,154.974
C02461=1062.038,-32.156,-65.507,171.701,26.758,154.974
C02462=1062.033,-32.405,-65.493,171.699,26.756,154.974
C02463=1062.027,-32.655,-65.480,171.698,26.754,154.973
C02464=1062.020,-32.905,-65.467,171.696,26.752,154.973
C02465=1062.014,-33.154,-65.453,171.695,26.750,154.973
C02466=1062.008,-33.404,-65.440,171.693,26.747,154.973
C02467=1062.002,-33.654,-65.428,171.691,26.746,154.973
C02468=1061.995,-33.931,-65.413,171.690,26.743,154.972
C02469=1061.988,-34.210,-65.398,171.688,26.741,154.972
C02470=1061.981,-34.488,-65.385,171.686,26.739,154.972
C02471=1061.975,-34.767,-65.370,171.684,26.736,154.972
C02472=1061.968,-35.016,-65.356,171.683,26.734,154.971
C02473=1061.962,-35.266,-65.344,171.681,26.732,154.971
C02474=1061.956,-35.516,-65.331,171.679,26.730,154.971
C02475=1061.950,-35.765,-65.318,171.678,26.728,154.971
C02476=1061.944,-36.015,-65.305,171.676,26.725,154.970
C02477=1061.938,-36.265,-65.292,171.675,26.724,154.970
C02478=1061.932,-36.514,-65.279,171.673,26.721,154.970
C02479=1061.926,-36.764,-65.266,171.672,26.719,154.970
C02480=1061.920,-37.013,-65.253,171.670,26.717,154.970
C02481=1061.914,-37.263,-65.241,171.668,26.715,154.969
C02482=1061.908,-37.512,-65.227,171.667,26.713,154.969
C02483=1061.902,-37.762,-65.215,171.665,26.711,154.969
C02484=1061.896,-38.011,-65.201,171.664,26.709,154.969
C02485=1061.890,-38.261,-65.189,171.662,26.706,154.968
C02486=1061.884,-38.511,-65.176,171.660,26.705,154.968
C02487=1061.878,-38.760,-65.163,171.659,26.702,154.968
C02488=1061.872,-39.010,-65.151,171.657,26.701,154.968
C02489=1061.865,-39.259,-65.137,171.656,26.698,154.968
C02490=1061.859,-39.509,-65.125,171.654,26.697,154.967
C02491=1061.853,-39.759,-65.113,171.653,26.694,154.967
C02492=1061.847,-40.008,-65.099,171.651,26.692,154.967
C02493=1061.841,-40.258,-65.087,171.649,26.690,154.967
C02494=1061.835,-40.507,-65.074,171.648,26.688,154.967
C02495=1061.828,-40.757,-65.062,171.646,26.686,154.966
C02496=1061.822,-41.007,-65.049,171.645,26.684,154.966
C02497=1061.816,-41.256,-65.036,171.643,26.682,154.966
C02498=1061.810,-41.506,-65.023,171.641,26.680,154.966
C02499=1061.804,-41.756,-65.011,171.640,26.678,154.966
C02500=1061.797,-42.005,-64.998,171.638,26.676,154.965
C02501=1061.791,-42.255,-64.986,171.637,26.674,154.965
C02502=1061.785,-42.505,-64.973,171.635,26.672,154.965
C02503=1061.779,-42.754,-64.960,171.633,26.670,154.965
C02504=1061.772,-43.003,-64.948,171.632,26.668,154.965
C02505=1061.766,-43.253,-64.935,171.630,26.666,154.964
C02506=1061.761,-43.503,-64.923,171.629,26.664,154.964
C02507=1061.754,-43.752,-64.909,171.627,26.662,154.964
C02508=1061.748,-44.002,-64.897,171.625,26.660,154.964
C02509=1061.742,-44.252,-64.885,171.624,26.658,154.963
C02510=1061.736,-44.502,-64.872,171.622,26.656,154.963
C02511=1061.730,-44.751,-64.859,171.620,26.654,154.963
C02512=1061.724,-45.001,-64.846,171.619,26.652,154.963
C02513=1061.717,-45.250,-64.835,171.617,26.650,154.963
C02514=1061.712,-45.500,-64.822,171.616,26.648,154.963
C02515=1061.706,-45.750,-64.810,171.614,26.646,154.962
C02516=1061.700,-45.999,-64.797,171.613,26.644,154.962
C02517=1061.693,-46.248,-64.785,171.611,26.642,154.962
C02518=1061.687,-46.498,-64.772,171.609,26.641,154.962
C02519=1061.681,-46.748,-64.759,171.608,26.638,154.962
C02520=1061.675,-46.998,-64.747,171.606,26.637,154.961
C02521=1061.668,-47.247,-64.734,171.605,26.634,154.961
C02522=1061.662,-47.497,-64.722,171.603,26.633,154.961
C02523=1061.657,-47.746,-64.709,171.601,26.631,154.961
C02524=1061.651,-47.996,-64.698,171.600,26.628,154.961
C02525=1061.645,-48.245,-64.685,171.598,26.627,154.960
C02526=1061.639,-48.495,-64.672,171.597,26.624,154.960
C02527=1061.633,-48.745,-64.660,171.595,26.623,154.960
C02528=1061.626,-48.995,-64.648,171.593,26.621,154.960
C02529=1061.621,-49.244,-64.636,171.592,26.619,154.960
C02530=1061.615,-49.493,-64.622,171.590,26.617,154.959
C02531=1061.608,-49.743,-64.610,171.588,26.615,154.959
C02532=1061.602,-50.022,-64.596,171.586,26.613,154.959
C02533=1061.595,-50.301,-64.583,171.584,26.610,154.959
C02534=1061.588,-50.580,-64.569,171.583,26.609,154.959
C02535=1061.580,-50.859,-64.555,171.580,26.606,154.959
C02536=1061.574,-51.108,-64.543,171.579,26.604,154.958
C02537=1061.569,-51.357,-64.531,171.577,26.603,154.958
C02538=1061.562,-51.607,-64.519,171.575,26.601,154.958
C02539=1061.556,-51.857,-64.506,171.574,26.599,154.958
C02540=1061.549,-52.106,-64.494,171.572,26.597,154.958
C02541=1061.543,-52.356,-64.482,171.570,26.595,154.958
C02542=1061.537,-52.606,-64.470,171.569,26.593,154.957
C02543=1061.530,-52.856,-64.459,171.567,26.592,154.957
C02544=1061.525,-53.105,-64.446,171.565,26.590,154.957
C02545=1061.518,-53.355,-64.434,171.564,26.588,154.957
C02546=1061.512,-53.604,-64.423,171.562,26.586,154.957
C02547=1061.506,-53.854,-64.410,171.561,26.584,154.957
C02548=1061.499,-54.104,-64.398,171.559,26.582,154.956
C02549=1061.493,-54.354,-64.385,171.557,26.581,154.956
C02550=1061.487,-54.603,-64.373,171.556,26.579,154.956
C02551=1061.481,-54.852,-64.362,171.554,26.577,154.956
C02552=1061.475,-55.102,-64.349,171.552,26.575,154.956
C02553=1061.468,-55.352,-64.337,171.551,26.574,154.956
C02554=1061.462,-55.602,-64.325,171.549,26.572,154.956
C02555=1061.456,-55.852,-64.314,171.548,26.570,154.955
C02556=1061.450,-56.101,-64.302,171.546,26.568,154.955
C02557=1061.444,-56.350,-64.289,171.544,26.566,154.955
C02558=1061.437,-56.600,-64.277,171.543,26.564,154.955
C02559=1061.431,-56.850,-64.266,171.541,26.563,154.955
C02560=1061.425,-57.100,-64.253,171.539,26.561,154.955
C02561=1061.419,-57.348,-64.241,171.538,26.559,154.954
C02562=1061.412,-57.599,-64.230,171.536,26.557,154.954
C02563=1061.406,-57.848,-64.218,171.534,26.556,154.954
C02564=1061.400,-58.098,-64.206,171.532,26.554,154.954
C02565=1061.394,-58.347,-64.193,171.530,26.552,154.954
C02566=1061.388,-58.597,-64.181,171.529,26.550,154.954
C02567=1061.381,-58.847,-64.170,171.527,26.548,154.953
C02568=1061.376,-59.097,-64.158,171.525,26.546,154.953
C02569=1061.370,-59.346,-64.146,171.524,26.544,154.953
C02570=1061.363,-59.595,-64.134,171.522,26.543,154.953
C02571=1061.357,-59.846,-64.122,171.520,26.541,154.953
C02572=1061.351,-60.095,-64.110,171.519,26.539,154.953
C02573=1061.345,-60.344,-64.099,171.517,26.538,154.953
C02574=1061.339,-60.594,-64.086,171.515,26.536,154.952
C02575=1061.332,-60.844,-64.075,171.514,26.534,154.952
C02576=1061.326,-61.093,-64.063,171.512,26.532,154.952
C02577=1061.320,-61.343,-64.051,171.511,26.531,154.952
C02578=1061.314,-61.593,-64.039,171.509,26.529,154.952
C02579=1061.307,-61.843,-64.028,171.507,26.527,154.952
C02580=1061.301,-62.092,-64.016,171.506,26.525,154.952
C02581=1061.295,-62.342,-64.003,171.504,26.524,154.951
C02582=1061.289,-62.592,-63.992,171.502,26.522,154.951
C02583=1061.283,-62.841,-63.981,171.501,26.520,154.951
C02584=1061.277,-63.091,-63.968,171.499,26.518,154.951
C02585=1061.271,-63.341,-63.957,171.497,26.517,154.951
C02586=1061.265,-63.590,-63.945,171.496,26.515,154.951
C02587=1061.259,-63.840,-63.933,171.494,26.513,154.951
C02588=1061.253,-64.090,-63.921,171.492,26.511,154.951
C02589=1061.246,-64.339,-63.910,171.490,26.509,154.950
C02590=1061.240,-64.589,-63.899,171.488,26.508,154.950
C02591=1061.235,-64.838,-63.886,171.487,26.506,154.950
C02592=1061.228,-65.087,-63.874,171.485,26.504,154.950
C02593=1061.222,-65.338,-63.863,171.483,26.503,154.950
C02594=1061.217,-65.587,-63.851,171.482,26.501,154.950
C02595=1061.210,-65.837,-63.840,171.480,26.500,154.950
C02596=1061.203,-66.117,-63.827,171.478,26.497,154.949
C02597=1061.196,-66.396,-63.814,171.477,26.496,154.949
C02598=1061.189,-66.677,-63.801,171.474,26.494,154.949
C02599=1061.183,-66.957,-63.787,171.472,26.492,154.949
C02600=1061.177,-67.208,-63.776,171.471,26.490,154.949
C02601=1061.171,-67.456,-63.764,171.469,26.488,154.949
C02602=1061.164,-67.706,-63.752,171.468,26.487,154.949
C02603=1061.159,-67.956,-63.741,171.466,26.485,154.948
C02604=1061.152,-68.205,-63.729,171.464,26.483,154.948
C02605=1061.147,-68.455,-63.718,171.463,26.481,154.948
C02606=1061.140,-68.705,-63.707,171.461,26.480,154.948
C02607=1061.134,-68.954,-63.695,171.459,26.478,154.948
C02608=1061.129,-69.204,-63.683,171.458,26.477,154.948
C02609=1061.122,-69.454,-63.671,171.456,26.475,154.948
C02610=1061.116,-69.704,-63.660,171.453,26.473,154.948
C02611=1061.110,-69.953,-63.649,171.452,26.471,154.947
C02612=1061.105,-70.203,-63.637,171.450,26.470,154.947
C02613=1061.098,-70.452,-63.625,171.448,26.468,154.947
C02614=1061.092,-70.702,-63.614,171.447,26.467,154.947
C02615=1061.086,-70.952,-63.603,171.445,26.465,154.947
C02616=1061.081,-71.201,-63.591,171.443,26.463,154.947
C02617=1061.074,-71.452,-63.580,171.442,26.461,154.947
C02618=1061.068,-71.700,-63.568,171.440,26.460,154.947
C02619=1061.062,-71.951,-63.557,171.438,26.458,154.946
C02620=1061.056,-72.200,-63.546,171.437,26.456,154.946
C02621=1061.050,-72.450,-63.533,171.435,26.455,154.946
C02622=1061.044,-72.699,-63.522,171.433,26.453,154.946
C02623=1061.038,-72.949,-63.510,171.432,26.452,154.946
C02624=1061.032,-73.199,-63.500,171.430,26.450,154.946
C02625=1061.026,-73.449,-63.488,171.428,26.448,154.946
C02626=1061.020,-73.698,-63.476,171.427,26.447,154.946
C02627=1061.014,-73.948,-63.465,171.425,26.445,154.946
C02628=1061.008,-74.198,-63.454,171.423,26.443,154.945
C02629=1061.002,-74.448,-63.443,171.422,26.442,154.945
C02630=1060.996,-74.697,-63.431,171.419,26.440,154.945
C02631=1060.990,-74.947,-63.420,171.417,26.439,154.945
C02632=1060.984,-75.196,-63.409,171.416,26.437,154.945
C02633=1060.977,-75.446,-63.397,171.414,26.436,154.945
C02634=1060.971,-75.695,-63.386,171.412,26.434,154.945
C02635=1060.964,-75.945,-63.376,171.411,26.433,154.945
C02636=1060.959,-76.195,-63.365,171.409,26.431,154.945
C02637=1060.952,-76.445,-63.353,171.407,26.429,154.945
C02638=1060.946,-76.694,-63.342,171.406,26.428,154.945
C02639=1060.941,-76.943,-63.331,171.404,26.426,154.944
C02640=1060.934,-77.194,-63.320,171.402,26.425,154.944
C02641=1060.928,-77.443,-63.309,171.401,26.423,154.944
C02642=1060.922,-77.693,-63.297,171.399,26.422,154.944
C02643=1060.916,-77.942,-63.286,171.397,26.421,154.944
C02644=1060.910,-78.192,-63.275,171.396,26.419,154.944
C02645=1060.904,-78.442,-63.264,171.394,26.418,154.944
C02646=1060.898,-78.692,-63.253,171.392,26.416,154.944
C02647=1060.892,-78.941,-63.242,171.389,26.414,154.944
C02648=1060.885,-79.191,-63.230,171.388,26.413,154.944
C02649=1060.880,-79.440,-63.219,171.386,26.411,154.944
C02650=1060.874,-79.690,-63.208,171.384,26.410,154.944
C02651=1060.867,-79.940,-63.197,171.383,26.408,154.943
C02652=1060.861,-80.189,-63.187,171.381,26.407,154.943
C02653=1060.855,-80.440,-63.175,171.379,26.406,154.943
C02654=1060.849,-80.689,-63.164,171.378,26.404,154.943
C02655=1060.842,-80.939,-63.154,171.376,26.403,154.943
C02656=1060.836,-81.188,-63.143,171.374,26.401,154.943
C02657=1060.830,-81.439,-63.132,171.372,26.400,154.943
C02658=1060.824,-81.687,-63.120,171.371,26.399,154.943
C02659=1060.817,-81.937,-63.109,171.369,26.397,154.943
C02660=1060.811,-82.220,-63.097,171.366,26.396,154.943
C02661=1060.803,-82.502,-63.085,171.365,26.394,154.943
C02662=1060.796,-82.785,-63.073,171.363,26.393,154.943
C02663=1060.789,-83.066,-63.061,171.360,26.391,154.943
C02664=1060.783,-83.316,-63.049,171.359,26.390,154.943
C02665=1060.777,-83.566,-63.039,171.357,26.388,154.942
C02666=1060.771,-83.815,-63.028,171.355,26.387,154.942
C02667=1060.764,-84.065,-63.017,171.354,26.385,154.942
C02668=1060.758,-84.315,-63.006,171.352,26.384,154.942
C02669=1060.752,-84.565,-62.995,171.350,26.383,154.942
C02670=1060.745,-84.814,-62.985,171.348,26.381,154.942
C02671=1060.740,-85.064,-62.974,171.347,26.380,154.942
C02672=1060.733,-85.314,-62.962,171.345,26.379,154.942
C02673=1060.727,-85.563,-62.952,171.343,26.377,154.942
C02674=1060.721,-85.813,-62.941,171.342,26.376,154.942
C02675=1060.715,-86.063,-62.930,171.340,26.374,154.942
C02676=1060.709,-86.313,-62.921,171.338,26.373,154.942
C02677=1060.702,-86.563,-62.909,171.336,26.371,154.942
C02678=1060.697,-86.812,-62.898,171.334,26.370,154.942
C02679=1060.690,-87.061,-62.888,171.332,26.369,154.942
C02680=1060.684,-87.312,-62.877,171.330,26.368,154.942
C02681=1060.678,-87.561,-62.866,171.329,26.366,154.942
C02682=1060.672,-87.810,-62.856,171.327,26.365,154.942
C02683=1060.665,-88.060,-62.844,171.325,26.364,154.942
C02684=1060.659,-88.310,-62.834,171.323,26.363,154.941
C02685=1060.653,-88.560,-62.824,171.322,26.361,154.941
C02686=1060.647,-88.810,-62.813,171.320,26.360,154.941
C02687=1060.641,-89.059,-62.802,171.318,26.359,154.941
C02688=1060.635,-89.309,-62.792,171.316,26.357,154.941
C02689=1060.629,-89.558,-62.781,171.315,26.356,154.941
C02690=1060.623,-89.808,-62.769,171.313,26.354,154.941
C02691=1060.616,-90.058,-62.760,171.311,26.353,154.941
C02692=1060.611,-90.308,-62.749,171.309,26.352,154.941
C02693=1060.604,-90.558,-62.738,171.307,26.350,154.941
C02694=1060.598,-90.807,-62.728,171.305,26.349,154.941
C02695=1060.592,-91.056,-62.717,171.303,26.348,154.941
C02696=1060.586,-91.306,-62.707,171.302,26.347,154.941
C02697=1060.580,-91.556,-62.696,171.300,26.345,154.941
C02698=1060.574,-91.806,-62.685,171.298,26.344,154.941
C02699=1060.567,-92.055,-62.675,171.297,26.343,154.941
C02700=1060.562,-92.305,-62.665,171.295,26.341,154.941
C02701=1060.556,-92.555,-62.653,171.293,26.340,154.941
C02702=1060.549,-92.805,-62.643,171.291,26.339,154.941
C02703=1060.543,-93.054,-62.632,171.290,26.338,154.941
C02704=1060.537,-93.304,-62.623,171.288,26.336,154.941
C02705=1060.532,-93.553,-62.612,171.286,26.335,154.941
C02706=1060.525,-93.804,-62.600,171.284,26.334,154.940
C02707=1060.519,-94.053,-62.591,171.282,26.332,154.941
C02708=1060.513,-94.303,-62.580,171.280,26.331,154.940
C02709=1060.507,-94.552,-62.570,171.278,26.330,154.940
C02710=1060.501,-94.803,-62.559,171.276,26.329,154.940
C02711=1060.494,-95.052,-62.549,171.275,26.328,154.940
C02712=1060.489,-95.301,-62.538,171.273,26.326,154.940
C02713=1060.483,-95.552,-62.528,171.271,26.325,154.940
C02714=1060.477,-95.801,-62.518,171.270,26.324,154.940
C02715=1060.471,-96.050,-62.507,171.268,26.323,154.940
C02716=1060.464,-96.301,-62.497,171.266,26.321,154.940
C02717=1060.458,-96.550,-62.486,171.264,26.320,154.940
C02718=1060.452,-96.800,-62.476,171.263,26.319,154.940
C02719=1060.447,-97.050,-62.465,171.261,26.318,154.940
C02720=1060.441,-97.299,-62.455,171.259,26.317,154.940
C02721=1060.435,-97.549,-62.445,171.257,26.316,154.940
C02722=1060.428,-97.799,-62.434,171.256,26.314,154.940
C02723=1060.422,-98.049,-62.424,171.253,26.313,154.940
C02724=1060.415,-98.333,-62.413,171.251,26.312,154.940
C02725=1060.408,-98.618,-62.401,171.249,26.311,154.940
C02726=1060.401,-98.902,-62.389,171.247,26.309,154.940
C02727=1060.394,-99.187,-62.378,171.245,26.308,154.940
C02728=1060.388,-99.436,-62.367,171.243,26.307,154.940
C02729=1060.382,-99.686,-62.357,171.241,26.306,154.940
C02730=1060.375,-99.936,-62.347,171.240,26.305,154.940
C02731=1060.369,-100.186,-62.336,171.238,26.303,154.940
C02732=1060.363,-100.435,-62.326,171.236,26.302,154.940
C02733=1060.357,-100.685,-62.317,171.234,26.302,154.940
C02734=1060.351,-100.935,-62.306,171.233,26.300,154.940
C02735=1060.345,-101.184,-62.296,171.230,26.299,154.940
C02736=1060.339,-101.434,-62.287,171.228,26.298,154.940
C02737=1060.332,-101.684,-62.275,171.226,26.297,154.940
C02738=1060.326,-101.934,-62.266,171.225,26.296,154.940
C02739=1060.320,-102.183,-62.255,171.223,26.294,154.940
C02740=1060.314,-102.433,-62.245,171.221,26.294,154.940
C02741=1060.308,-102.683,-62.235,171.219,26.293,154.940
C02742=1060.301,-102.932,-62.225,171.217,26.292,154.940
C02743=1060.296,-103.182,-62.215,171.216,26.290,154.940
C02744=1060.290,-103.432,-62.205,171.214,26.289,154.940
C02745=1060.283,-103.681,-62.195,171.212,26.289,154.940
C02746=1060.277,-103.932,-62.184,171.210,26.287,154.940
C02747=1060.271,-104.181,-62.175,171.209,26.286,154.940
C02748=1060.265,-104.431,-62.165,171.207,26.285,154.940
C02749=1060.258,-104.680,-62.155,171.205,26.285,154.940
C02750=1060.253,-104.931,-62.145,171.202,26.283,154.940
C02751=1060.247,-105.180,-62.135,171.201,26.282,154.940
C02752=1060.240,-105.429,-62.125,171.199,26.281,154.940
C02753=1060.234,-105.679,-62.115,171.197,26.280,154.940
C02754=1060.229,-105.929,-62.105,171.195,26.279,154.940
C02755=1060.222,-106.179,-62.095,171.193,26.278,154.940
C02756=1060.216,-106.428,-62.085,171.192,26.277,154.940
C02757=1060.210,-106.678,-62.076,171.190,26.276,154.940
C02758=1060.204,-106.928,-62.065,171.188,26.275,154.940
C02759=1060.198,-107.177,-62.055,171.186,26.274,154.940
C02760=1060.192,-107.427,-62.046,171.184,26.273,154.940
C02761=1060.185,-107.677,-62.036,171.183,26.272,154.940
C02762=1060.178,-107.927,-62.025,171.181,26.271,154.940
C02763=1060.173,-108.177,-62.015,171.179,26.270,154.940
C02764=1060.167,-108.427,-62.006,171.176,26.269,154.940
C02765=1060.161,-108.677,-61.996,171.174,26.268,154.941
C02766=1060.154,-108.926,-61.986,171.173,26.267,154.941
C02767=1060.148,-109.176,-61.976,171.171,26.266,154.941
C02768=1060.142,-109.425,-61.967,171.169,26.265,154.941
C02769=1060.136,-109.675,-61.957,171.167,26.264,154.941
C02770=1060.129,-109.925,-61.948,171.165,26.264,154.941
C02771=1060.124,-110.174,-61.937,171.164,26.263,154.941
C02772=1060.118,-110.424,-61.927,171.162,26.262,154.941
C02773=1060.111,-110.674,-61.917,171.160,26.261,154.941
C02774=1060.105,-110.924,-61.908,171.158,26.260,154.941
C02775=1060.099,-111.174,-61.898,171.156,26.259,154.941
C02776=1060.093,-111.423,-61.889,171.155,26.259,154.941
C02777=1060.086,-111.673,-61.879,171.153,26.257,154.941
C02778=1060.080,-111.922,-61.869,171.151,26.256,154.941
C02779=1060.074,-112.172,-61.859,171.148,26.255,154.941
C02780=1060.068,-112.422,-61.850,171.147,26.254,154.941
C02781=1060.062,-112.672,-61.840,171.145,26.254,154.941
C02782=1060.056,-112.922,-61.830,171.143,26.252,154.941
C02783=1060.050,-113.172,-61.821,171.141,26.252,154.941
C02784=1060.044,-113.422,-61.811,171.139,26.251,154.941
C02785=1060.038,-113.671,-61.801,171.137,26.250,154.941
C02786=1060.031,-113.921,-61.791,171.136,26.250,154.941
C02787=1060.025,-114.170,-61.782,171.134,26.248,154.941
C02788=1060.019,-114.453,-61.771,171.132,26.248,154.941
C02789=1060.011,-114.737,-61.761,171.129,26.246,154.942
C02790=1060.005,-115.019,-61.749,171.127,26.246,154.942
C02791=1059.998,-115.302,-61.738,171.126,26.245,154.942
C02792=1059.992,-115.552,-61.729,171.124,26.244,154.942
C02793=1059.985,-115.802,-61.719,171.121,26.243,154.942
C02794=1059.979,-116.052,-61.710,171.119,26.242,154.942
C02795=1059.972,-116.301,-61.701,171.117,26.241,154.942
C02796=1059.966,-116.551,-61.691,171.116,26.240,154.942
C02797=1059.961,-116.800,-61.682,171.114,26.240,154.942
C02798=1059.954,-117.050,-61.672,171.112,26.239,154.942
C02799=1059.948,-117.300,-61.663,171.110,26.238,154.942
C02800=1059.942,-117.550,-61.653,171.108,26.237,154.942
C02801=1059.936,-117.799,-61.644,171.106,26.237,154.942
C02802=1059.930,-118.049,-61.634,171.105,26.236,154.942
C02803=1059.924,-118.299,-61.624,171.103,26.235,154.942
C02804=1059.917,-118.549,-61.615,171.101,26.235,154.942
C02805=1059.911,-118.799,-61.605,171.099,26.234,154.943
C02806=1059.905,-119.048,-61.596,171.097,26.233,154.943
C02807=1059.899,-119.298,-61.586,171.095,26.232,154.943
C02808=1059.894,-119.548,-61.578,171.093,26.232,154.943
C02809=1059.887,-119.798,-61.568,171.091,26.231,154.943
C02810=1059.881,-120.047,-61.559,171.089,26.230,154.943
C02811=1059.874,-120.297,-61.550,171.087,26.229,154.943
C02812=1059.868,-120.547,-61.540,171.085,26.228,154.943
C02813=1059.862,-120.797,-61.530,171.083,26.228,154.943
C02814=1059.856,-121.046,-61.521,171.082,26.227,154.943
C02815=1059.850,-121.295,-61.512,171.080,26.226,154.943
C02816=1059.844,-121.546,-61.503,171.078,26.226,154.943
C02817=1059.838,-121.796,-61.493,171.076,26.225,154.943
C02818=1059.831,-122.045,-61.484,171.074,26.224,154.944
C02819=1059.825,-122.295,-61.475,171.072,26.223,154.944
C02820=1059.819,-122.545,-61.465,171.070,26.223,154.944
C02821=1059.813,-122.795,-61.456,171.069,26.222,154.944
C02822=1059.808,-123.044,-61.447,171.067,26.222,154.944
C02823=1059.801,-123.294,-61.438,171.065,26.221,154.944
C02824=1059.794,-123.544,-61.429,171.063,26.220,154.944
C02825=1059.788,-123.793,-61.419,171.060,26.220,154.944
C02826=1059.782,-124.044,-61.410,171.058,26.218,154.944
C02827=1059.777,-124.293,-61.401,171.057,26.218,154.944
C02828=1059.771,-124.543,-61.391,171.055,26.217,154.944
C02829=1059.764,-124.792,-61.382,171.053,26.217,154.944
C02830=1059.758,-125.043,-61.374,171.051,26.216,154.945
C02831=1059.752,-125.292,-61.364,171.049,26.216,154.945
C02832=1059.746,-125.542,-61.354,171.047,26.215,154.945
C02833=1059.739,-125.791,-61.346,171.045,26.214,154.945
C02834=1059.733,-126.041,-61.337,171.043,26.214,154.945
C02835=1059.727,-126.291,-61.327,171.042,26.213,154.945
C02836=1059.721,-126.541,-61.318,171.040,26.213,154.945
C02837=1059.714,-126.791,-61.310,171.038,26.212,154.945
C02838=1059.709,-127.040,-61.300,171.036,26.212,154.945
C02839=1059.703,-127.290,-61.291,171.034,26.211,154.945
C02840=1059.696,-127.540,-61.283,171.032,26.210,154.946
C02841=1059.690,-127.790,-61.273,171.030,26.210,154.946
C02842=1059.685,-128.039,-61.263,171.028,26.208,154.946
C02843=1059.681,-128.290,-61.253,171.027,26.207,154.946
C02844=1059.679,-128.540,-61.242,171.025,26.205,154.945
C02845=1059.677,-128.791,-61.230,171.024,26.203,154.945
C02846=1059.677,-129.041,-61.218,171.023,26.199,154.945
C02847=1059.679,-129.291,-61.205,171.021,26.196,154.944
C02848=1059.681,-129.543,-61.191,171.020,26.191,154.943
C02849=1059.686,-129.794,-61.177,171.020,26.186,154.943
C02850=1059.692,-130.045,-61.161,171.019,26.181,154.942
C02851=1059.699,-130.296,-61.145,171.020,26.174,154.941
C02852=1059.321,-130.318,-61.342,170.972,26.334,154.974
C02853=1059.314,-130.069,-61.358,170.972,26.340,154.975
C02854=1059.309,-129.818,-61.373,170.972,26.346,154.976
C02855=1059.303,-129.567,-61.388,170.973,26.351,154.977
C02856=1059.301,-129.314,-61.402,170.974,26.355,154.977
C02857=1059.299,-129.064,-61.415,170.975,26.359,154.978
C02858=1059.299,-128.814,-61.426,170.976,26.362,154.978
C02859=1059.300,-128.563,-61.439,170.978,26.365,154.979
C02860=1059.303,-128.312,-61.449,170.979,26.367,154.979
C02861=1059.306,-128.062,-61.460,170.981,26.368,154.979
C02862=1059.312,-127.813,-61.469,170.983,26.369,154.979
C02863=1059.318,-127.563,-61.478,170.984,26.370,154.979
C02864=1059.324,-127.313,-61.488,170.986,26.371,154.979
C02865=1059.330,-127.063,-61.497,170.988,26.371,154.979
C02866=1059.336,-126.814,-61.505,170.990,26.372,154.979
C02867=1059.342,-126.564,-61.515,170.992,26.372,154.978
C02868=1059.348,-126.314,-61.524,170.994,26.373,154.978
C02869=1059.355,-126.064,-61.533,170.996,26.373,154.978
C02870=1059.361,-125.814,-61.542,170.998,26.374,154.978
C02871=1059.367,-125.565,-61.552,170.999,26.374,154.978
C02872=1059.373,-125.315,-61.560,171.001,26.375,154.978
C02873=1059.380,-125.065,-61.569,171.003,26.376,154.978
C02874=1059.386,-124.816,-61.579,171.005,26.376,154.978
C02875=1059.392,-124.566,-61.589,171.007,26.377,154.978
C02876=1059.398,-124.315,-61.597,171.009,26.377,154.978
C02877=1059.404,-124.067,-61.606,171.012,26.378,154.977
C02878=1059.410,-123.817,-61.616,171.013,26.379,154.977
C02879=1059.416,-123.567,-61.625,171.015,26.380,154.977
C02880=1059.422,-123.316,-61.634,171.017,26.380,154.977
C02881=1059.429,-123.067,-61.644,171.019,26.381,154.977
C02882=1059.434,-122.818,-61.653,171.021,26.382,154.977
C02883=1059.441,-122.568,-61.662,171.023,26.382,154.977
C02884=1059.447,-122.318,-61.671,171.025,26.383,154.977
C02885=1059.453,-122.068,-61.680,171.026,26.383,154.977
C02886=1059.459,-121.818,-61.690,171.028,26.384,154.977
C02887=1059.465,-121.568,-61.699,171.030,26.385,154.977
C02888=1059.471,-121.319,-61.708,171.032,26.386,154.977
C02889=1059.477,-121.069,-61.718,171.034,26.386,154.976
C02890=1059.484,-120.820,-61.727,171.036,26.387,154.976
C02891=1059.490,-120.570,-61.736,171.037,26.388,154.976
C02892=1059.496,-120.320,-61.745,171.040,26.389,154.976
C02893=1059.502,-120.070,-61.755,171.042,26.389,154.976
C02894=1059.508,-119.820,-61.765,171.044,26.390,154.976
C02895=1059.515,-119.570,-61.774,171.046,26.391,154.976
C02896=1059.520,-119.321,-61.783,171.048,26.391,154.976
C02897=1059.526,-119.071,-61.793,171.049,26.392,154.976
C02898=1059.533,-118.822,-61.802,171.051,26.393,154.976
C02899=1059.539,-118.572,-61.812,171.053,26.394,154.976
C02900=1059.546,-118.322,-61.821,171.055,26.394,154.976
C02901=1059.552,-118.073,-61.831,171.057,26.395,154.976
C02902=1059.558,-117.823,-61.840,171.059,26.395,154.975
C02903=1059.564,-117.572,-61.849,171.060,26.397,154.975
C02904=1059.570,-117.323,-61.859,171.062,26.397,154.975
C02905=1059.576,-117.073,-61.868,171.064,26.398,154.975
C02906=1059.582,-116.824,-61.877,171.067,26.399,154.975
C02907=1059.588,-116.574,-61.887,171.069,26.400,154.975
C02908=1059.594,-116.324,-61.896,171.071,26.400,154.975
C02909=1059.600,-116.074,-61.906,171.072,26.401,154.975
C02910=1059.606,-115.824,-61.916,171.074,26.402,154.975
C02911=1059.613,-115.575,-61.925,171.076,26.403,154.975
C02912=1059.619,-115.325,-61.935,171.078,26.404,154.975
C02913=1059.626,-115.042,-61.946,171.080,26.404,154.975
C02914=1059.633,-114.759,-61.956,171.083,26.406,154.975
C02915=1059.640,-114.476,-61.967,171.084,26.406,154.975
C02916=1059.647,-114.193,-61.979,171.086,26.407,154.975
C02917=1059.653,-113.943,-61.989,171.088,26.408,154.975
C02918=1059.659,-113.693,-61.998,171.090,26.409,154.974
C02919=1059.665,-113.443,-62.008,171.093,26.410,154.974
C02920=1059.671,-113.194,-62.017,171.094,26.411,154.974
C02921=1059.677,-112.944,-62.027,171.096,26.412,154.974
C02922=1059.683,-112.695,-62.036,171.098,26.412,154.974
C02923=1059.690,-112.445,-62.046,171.100,26.413,154.974
C02924=1059.696,-112.195,-62.055,171.102,26.414,154.974
C02925=1059.702,-111.946,-62.066,171.103,26.415,154.974
C02926=1059.708,-111.696,-62.075,171.105,26.416,154.974
C02927=1059.714,-111.446,-62.085,171.107,26.417,154.974
C02928=1059.720,-111.196,-62.095,171.109,26.417,154.974
C02929=1059.726,-110.946,-62.104,171.111,26.419,154.974
C02930=1059.732,-110.697,-62.114,171.113,26.419,154.974
C02931=1059.739,-110.447,-62.124,171.114,26.420,154.974
C02932=1059.745,-110.198,-62.134,171.116,26.421,154.974
C02933=1059.751,-109.948,-62.143,171.119,26.422,154.974
C02934=1059.757,-109.698,-62.153,171.121,26.423,154.974
C02935=1059.763,-109.448,-62.163,171.123,26.424,154.974
C02936=1059.769,-109.198,-62.173,171.124,26.425,154.974
C02937=1059.775,-108.949,-62.183,171.126,26.426,154.974
C02938=1059.782,-108.698,-62.193,171.128,26.427,154.974
C02939=1059.788,-108.449,-62.202,171.130,26.427,154.974
C02940=1059.795,-108.199,-62.212,171.132,26.429,154.974
C02941=1059.801,-107.950,-62.222,171.133,26.430,154.974
C02942=1059.807,-107.700,-62.232,171.135,26.430,154.974
C02943=1059.813,-107.450,-62.241,171.137,26.432,154.974
C02944=1059.819,-107.200,-62.252,171.139,26.433,154.974
C02945=1059.825,-106.951,-62.262,171.141,26.433,154.973
C02946=1059.831,-106.701,-62.271,171.143,26.435,154.973
C02947=1059.838,-106.451,-62.281,171.145,26.436,154.973
C02948=1059.843,-106.202,-62.292,171.147,26.436,154.973
C02949=1059.850,-105.952,-62.301,171.149,26.438,154.973
C02950=1059.856,-105.702,-62.311,171.150,26.439,154.973
C02951=1059.862,-105.453,-62.321,171.152,26.439,154.973
C02952=1059.868,-105.203,-62.331,171.154,26.440,154.973
C02953=1059.874,-104.953,-62.341,171.156,26.442,154.973
C02954=1059.880,-104.704,-62.351,171.158,26.443,154.973
C02955=1059.886,-104.453,-62.362,171.159,26.443,154.973
C02956=1059.892,-104.203,-62.371,171.161,26.444,154.973
C02957=1059.899,-103.954,-62.382,171.163,26.446,154.973
C02958=1059.905,-103.704,-62.391,171.165,26.447,154.973
C02959=1059.911,-103.454,-62.401,171.167,26.447,154.973
C02960=1059.917,-103.205,-62.412,171.169,26.449,154.973
C02961=1059.923,-102.955,-62.421,171.171,26.450,154.973
C02962=1059.929,-102.706,-62.432,171.173,26.451,154.973
C02963=1059.935,-102.456,-62.442,171.175,26.452,154.973
C02964=1059.942,-102.207,-62.452,171.176,26.453,154.973
C02965=1059.948,-101.956,-62.463,171.178,26.454,154.973
C02966=1059.954,-101.706,-62.472,171.180,26.455,154.973
C02967=1059.960,-101.457,-62.482,171.182,26.456,154.973
C02968=1059.966,-101.207,-62.493,171.183,26.457,154.973
C02969=1059.972,-100.958,-62.503,171.185,26.459,154.973
C02970=1059.978,-100.708,-62.512,171.187,26.459,154.973
C02971=1059.984,-100.458,-62.523,171.189,26.460,154.973
C02972=1059.991,-100.208,-62.533,171.191,26.461,154.973
C02973=1059.997,-99.959,-62.544,171.192,26.463,154.973
C02974=1060.003,-99.708,-62.554,171.195,26.464,154.973
C02975=1060.009,-99.459,-62.564,171.197,26.465,154.973
C02976=1060.015,-99.209,-62.574,171.199,26.466,154.973
C02977=1060.022,-98.925,-62.585,171.200,26.467,154.973
C02978=1060.029,-98.640,-62.597,171.202,26.469,154.973
C02979=1060.037,-98.355,-62.609,171.205,26.470,154.973
C02980=1060.044,-98.071,-62.621,171.207,26.471,154.973
C02981=1060.050,-97.821,-62.631,171.208,26.472,154.973
C02982=1060.056,-97.571,-62.641,171.210,26.473,154.973
C02983=1060.062,-97.321,-62.651,171.212,26.475,154.973
C02984=1060.067,-97.072,-62.662,171.214,26.476,154.973
C02985=1060.075,-96.822,-62.673,171.215,26.477,154.973
C02986=1060.080,-96.572,-62.683,171.218,26.478,154.973
C02987=1060.086,-96.323,-62.693,171.220,26.480,154.973
C02988=1060.092,-96.073,-62.704,171.222,26.481,154.973
C02989=1060.098,-95.823,-62.714,171.223,26.482,154.973
C02990=1060.104,-95.574,-62.724,171.225,26.483,154.973
C02991=1060.110,-95.323,-62.735,171.227,26.484,154.973
C02992=1060.117,-95.074,-62.745,171.229,26.485,154.973
C02993=1060.122,-94.825,-62.756,171.230,26.486,154.973
C02994=1060.129,-94.575,-62.766,171.232,26.488,154.974
C02995=1060.134,-94.325,-62.776,171.234,26.489,154.974
C02996=1060.141,-94.075,-62.788,171.236,26.490,154.974
C02997=1060.147,-93.825,-62.797,171.237,26.492,154.974
C02998=1060.153,-93.576,-62.808,171.239,26.493,154.974
C02999=1060.159,-93.327,-62.818,171.241,26.494,154.974
C03000=1060.165,-93.077,-62.829,171.244,26.495,154.974
C03001=1060.171,-92.826,-62.840,171.245,26.497,154.974
C03002=1060.177,-92.577,-62.850,171.247,26.498,154.974
C03003=1060.183,-92.328,-62.861,171.249,26.499,154.974
C03004=1060.189,-92.078,-62.871,171.250,26.501,154.974
C03005=1060.196,-91.828,-62.882,171.252,26.502,154.974
C03006=1060.201,-91.578,-62.893,171.254,26.503,154.974
C03007=1060.208,-91.329,-62.903,171.256,26.504,154.974
C03008=1060.213,-91.079,-62.914,171.257,26.506,154.974
C03009=1060.219,-90.829,-62.924,171.259,26.507,154.974
C03010=1060.226,-90.579,-62.935,171.261,26.508,154.974
C03011=1060.232,-90.330,-62.946,171.263,26.509,154.974
C03012=1060.239,-90.080,-62.956,171.264,26.510,154.974
C03013=1060.245,-89.831,-62.967,171.266,26.512,154.974
C03014=1060.250,-89.581,-62.977,171.268,26.513,154.974
C03015=1060.256,-89.331,-62.988,171.270,26.515,154.974
C03016=1060.263,-89.081,-62.999,171.272,26.516,154.974
C03017=1060.269,-88.832,-63.010,171.274,26.517,154.974
C03018=1060.275,-88.582,-63.020,171.276,26.519,154.975
C03019=1060.281,-88.332,-63.031,171.277,26.520,154.975
C03020=1060.287,-88.082,-63.041,171.279,26.521,154.975
C03021=1060.293,-87.833,-63.052,171.281,26.522,154.975
C03022=1060.300,-87.583,-63.063,171.283,26.524,154.975
C03023=1060.305,-87.333,-63.074,171.284,26.525,154.975
C03024=1060.312,-87.084,-63.084,171.286,26.526,154.975
C03025=1060.318,-86.834,-63.095,171.288,26.528,154.975
C03026=1060.324,-86.584,-63.106,171.290,26.529,154.975
C03027=1060.330,-86.335,-63.116,171.291,26.530,154.975
C03028=1060.337,-86.085,-63.128,171.293,26.531,154.975
C03029=1060.342,-85.836,-63.139,171.295,26.533,154.975
C03030=1060.349,-85.586,-63.149,171.297,26.535,154.975
C03031=1060.355,-85.336,-63.159,171.299,26.536,154.975
C03032=1060.361,-85.086,-63.170,171.301,26.537,154.975
C03033=1060.368,-84.836,-63.181,171.303,26.539,154.975
C03034=1060.374,-84.587,-63.192,171.304,26.540,154.975
C03035=1060.379,-84.337,-63.203,171.306,26.541,154.975
C03036=1060.386,-84.087,-63.213,171.308,26.543,154.975
C03037=1060.392,-83.838,-63.224,171.309,26.544,154.975
C03038=1060.398,-83.588,-63.235,171.311,26.546,154.976
C03039=1060.404,-83.338,-63.246,171.313,26.547,154.976
C03040=1060.411,-83.089,-63.257,171.315,26.548,154.976
C03041=1060.417,-82.806,-63.270,171.317,26.550,154.976
C03042=1060.425,-82.524,-63.282,171.319,26.551,154.976
C03043=1060.432,-82.242,-63.294,171.321,26.553,154.976
C03044=1060.438,-81.959,-63.306,171.323,26.554,154.976
C03045=1060.446,-81.710,-63.318,171.325,26.556,154.976
C03046=1060.451,-81.460,-63.329,171.327,26.557,154.976
C03047=1060.458,-81.210,-63.340,171.328,26.559,154.976
C03048=1060.464,-80.961,-63.350,171.330,26.560,154.976
C03049=1060.470,-80.711,-63.361,171.332,26.561,154.976
C03050=1060.476,-80.461,-63.372,171.334,26.563,154.976
C03051=1060.483,-80.211,-63.383,171.335,26.564,154.976
C03052=1060.489,-79.962,-63.394,171.337,26.566,154.977
C03053=1060.495,-79.712,-63.405,171.339,26.567,154.977
C03054=1060.501,-79.462,-63.416,171.340,26.569,154.977
C03055=1060.507,-79.213,-63.427,171.342,26.570,154.977
C03056=1060.513,-78.963,-63.439,171.344,26.571,154.977
C03057=1060.519,-78.714,-63.450,171.346,26.573,154.977
C03058=1060.526,-78.463,-63.461,171.348,26.575,154.977
C03059=1060.531,-78.214,-63.472,171.350,26.576,154.977
C03060=1060.538,-77.964,-63.483,171.352,26.578,154.977
C03061=1060.544,-77.715,-63.494,171.353,26.579,154.977
C03062=1060.549,-77.465,-63.505,171.355,26.580,154.977
C03063=1060.556,-77.215,-63.517,171.357,26.582,154.977
C03064=1060.562,-76.966,-63.527,171.358,26.583,154.977
C03065=1060.569,-76.716,-63.538,171.360,26.585,154.978
C03066=1060.575,-76.467,-63.550,171.362,26.586,154.978
C03067=1060.581,-76.217,-63.561,171.363,26.588,154.978
C03068=1060.587,-75.967,-63.572,171.365,26.590,154.978
C03069=1060.593,-75.717,-63.583,171.367,26.591,154.978
C03070=1060.599,-75.468,-63.595,171.368,26.593,154.978
C03071=1060.605,-75.218,-63.606,171.370,26.594,154.978
C03072=1060.611,-74.969,-63.617,171.372,26.595,154.978
C03073=1060.618,-74.718,-63.628,171.374,26.597,154.978
C03074=1060.624,-74.469,-63.640,171.375,26.598,154.978
C03075=1060.630,-74.219,-63.651,171.378,26.600,154.979
C03076=1060.636,-73.970,-63.662,171.380,26.602,154.979
C03077=1060.642,-73.720,-63.674,171.381,26.603,154.979
C03078=1060.647,-73.470,-63.685,171.383,26.605,154.979
C03079=1060.654,-73.220,-63.696,171.385,26.607,154.979
C03080=1060.660,-72.971,-63.708,171.386,26.608,154.979
C03081=1060.666,-72.721,-63.719,171.388,26.610,154.979
C03082=1060.672,-72.472,-63.730,171.390,26.611,154.979
C03083=1060.678,-72.222,-63.743,171.391,26.613,154.979
C03084=1060.683,-71.972,-63.754,171.393,26.615,154.980
C03085=1060.690,-71.723,-63.766,171.395,26.616,154.980
C03086=1060.696,-71.473,-63.776,171.396,26.618,154.980
C03087=1060.702,-71.223,-63.788,171.398,26.620,154.980
C03088=1060.707,-70.974,-63.800,171.400,26.621,154.980
C03089=1060.714,-70.724,-63.811,171.401,26.623,154.980
C03090=1060.720,-70.475,-63.823,171.403,26.625,154.980
C03091=1060.726,-70.225,-63.834,171.405,26.626,154.980
C03092=1060.732,-69.975,-63.845,171.406,26.628,154.981
C03093=1060.738,-69.725,-63.857,171.408,26.630,154.981
C03094=1060.744,-69.476,-63.868,171.410,26.631,154.981
C03095=1060.750,-69.226,-63.880,171.412,26.633,154.981
C03096=1060.757,-68.976,-63.891,171.414,26.635,154.981
C03097=1060.762,-68.727,-63.904,171.416,26.636,154.981
C03098=1060.768,-68.477,-63.915,171.417,26.638,154.981
C03099=1060.774,-68.228,-63.926,171.419,26.640,154.981
C03100=1060.781,-67.978,-63.938,171.421,26.642,154.982
C03101=1060.786,-67.728,-63.950,171.422,26.643,154.982
C03102=1060.792,-67.478,-63.961,171.424,26.645,154.982
C03103=1060.799,-67.229,-63.973,171.426,26.647,154.982
C03104=1060.805,-66.979,-63.984,171.427,26.648,154.982
C03105=1060.811,-66.699,-63.998,171.429,26.650,154.982
C03106=1060.818,-66.419,-64.011,171.431,26.652,154.982
C03107=1060.825,-66.138,-64.024,171.433,26.654,154.982
C03108=1060.832,-65.859,-64.037,171.435,26.656,154.983
C03109=1060.838,-65.609,-64.048,171.436,26.657,154.983
C03110=1060.844,-65.359,-64.060,171.438,26.659,154.983
C03111=1060.850,-65.110,-64.072,171.440,26.661,154.983
C03112=1060.856,-64.860,-64.083,171.441,26.663,154.983
C03113=1060.862,-64.610,-64.095,171.443,26.664,154.983
C03114=1060.868,-64.360,-64.107,171.445,26.666,154.983
C03115=1060.875,-64.111,-64.119,171.446,26.668,154.984
C03116=1060.881,-63.862,-64.130,171.448,26.669,154.984
C03117=1060.886,-63.611,-64.142,171.451,26.671,154.984
C03118=1060.893,-63.362,-64.154,171.452,26.673,154.984
C03119=1060.899,-63.113,-64.166,171.454,26.675,154.984
C03120=1060.905,-62.862,-64.177,171.456,26.677,154.984
C03121=1060.911,-62.613,-64.189,171.457,26.678,154.984
C03122=1060.917,-62.364,-64.201,171.459,26.680,154.985
C03123=1060.923,-62.113,-64.213,171.460,26.682,154.985
C03124=1060.930,-61.864,-64.225,171.462,26.684,154.985
C03125=1060.936,-61.615,-64.236,171.464,26.685,154.985
C03126=1060.942,-61.365,-64.248,171.465,26.687,154.985
C03127=1060.948,-61.115,-64.260,171.467,26.689,154.985
C03128=1060.954,-60.865,-64.272,171.469,26.691,154.985
C03129=1060.961,-60.616,-64.284,171.470,26.692,154.986
C03130=1060.966,-60.366,-64.296,171.472,26.694,154.986
C03131=1060.973,-60.116,-64.308,171.474,26.696,154.986
C03132=1060.979,-59.868,-64.319,171.475,26.697,154.986
C03133=1060.985,-59.618,-64.332,171.477,26.699,154.986
C03134=1060.991,-59.367,-64.343,171.479,26.701,154.986
C03135=1060.998,-59.118,-64.355,171.480,26.703,154.986
C03136=1061.003,-58.869,-64.367,171.482,26.704,154.987
C03137=1061.010,-58.619,-64.379,171.484,26.706,154.987
C03138=1061.016,-58.369,-64.390,171.485,26.708,154.987
C03139=1061.022,-58.119,-64.403,171.487,26.710,154.987
C03140=1061.028,-57.870,-64.414,171.489,26.711,154.987
C03141=1061.034,-57.620,-64.427,171.491,26.713,154.987
C03142=1061.041,-57.371,-64.439,171.493,26.715,154.987
C03143=1061.047,-57.121,-64.451,171.495,26.717,154.988
C03144=1061.053,-56.871,-64.463,171.496,26.718,154.988
C03145=1061.059,-56.622,-64.474,171.498,26.720,154.988
C03146=1061.065,-56.372,-64.486,171.499,26.722,154.988
C03147=1061.071,-56.122,-64.499,171.501,26.724,154.988
C03148=1061.078,-55.873,-64.511,171.503,26.726,154.988
C03149=1061.085,-55.623,-64.523,171.504,26.728,154.989
C03150=1061.090,-55.374,-64.535,171.506,26.729,154.989
C03151=1061.097,-55.124,-64.547,171.508,26.731,154.989
C03152=1061.102,-54.874,-64.559,171.509,26.733,154.989
C03153=1061.109,-54.624,-64.571,171.511,26.735,154.989
C03154=1061.116,-54.375,-64.583,171.513,26.736,154.989
C03155=1061.121,-54.125,-64.595,171.514,26.738,154.989
C03156=1061.127,-53.876,-64.607,171.516,26.740,154.990
C03157=1061.133,-53.626,-64.619,171.517,26.742,154.990
C03158=1061.140,-53.377,-64.631,171.519,26.744,154.990
C03159=1061.147,-53.127,-64.643,171.521,26.745,154.990
C03160=1061.153,-52.877,-64.656,171.522,26.747,154.990
C03161=1061.159,-52.628,-64.668,171.524,26.749,154.990
C03162=1061.165,-52.378,-64.680,171.526,26.751,154.991
C03163=1061.171,-52.129,-64.692,171.527,26.752,154.991
C03164=1061.178,-51.879,-64.704,171.529,26.755,154.991
C03165=1061.184,-51.629,-64.716,171.531,26.756,154.991
C03166=1061.190,-51.380,-64.728,171.532,26.758,154.991
C03167=1061.196,-51.130,-64.741,171.534,26.760,154.991
C03168=1061.203,-50.880,-64.753,171.536,26.762,154.991
C03169=1061.210,-50.601,-64.767,171.538,26.764,154.992
C03170=1061.217,-50.323,-64.780,171.540,26.766,154.992
C03171=1061.224,-50.044,-64.794,171.541,26.768,154.992
C03172=1061.230,-49.764,-64.808,171.543,26.770,154.992
C03173=1061.236,-49.516,-64.820,171.545,26.772,154.992
C03174=1061.242,-49.266,-64.833,171.547,26.774,154.993
C03175=1061.248,-49.016,-64.845,171.549,26.777,154.993
C03176=1061.254,-48.766,-64.858,171.550,26.778,154.993
C03177=1061.261,-48.516,-64.870,171.552,26.780,154.993
C03178=1061.267,-48.266,-64.882,171.554,26.782,154.993
C03179=1061.273,-48.017,-64.895,171.555,26.784,154.994
C03180=1061.279,-47.768,-64.907,171.557,26.786,154.994
C03181=1061.285,-47.518,-64.920,171.558,26.788,154.994
C03182=1061.291,-47.269,-64.932,171.560,26.790,154.994
C03183=1061.297,-47.019,-64.945,171.562,26.792,154.994
C03184=1061.303,-46.769,-64.957,171.563,26.794,154.995
C03185=1061.309,-46.519,-64.969,171.565,26.795,154.995
C03186=1061.316,-46.270,-64.982,171.566,26.798,154.995
C03187=1061.321,-46.020,-64.995,171.568,26.800,154.995
C03188=1061.327,-45.771,-65.007,171.570,26.802,154.995
C03189=1061.333,-45.521,-65.019,171.571,26.804,154.996
C03190=1061.339,-45.271,-65.032,171.573,26.806,154.996
C03191=1061.345,-45.022,-65.045,171.575,26.808,154.996
C03192=1061.352,-44.773,-65.057,171.576,26.809,154.996
C03193=1061.358,-44.523,-65.070,171.578,26.812,154.996
C03194=1061.364,-44.273,-65.082,171.579,26.813,154.996
C03195=1061.370,-44.024,-65.095,171.581,26.816,154.997
C03196=1061.377,-43.774,-65.107,171.583,26.817,154.997
C03197=1061.383,-43.524,-65.120,171.584,26.820,154.997
C03198=1061.389,-43.274,-65.132,171.586,26.821,154.997
C03199=1061.395,-43.025,-65.146,171.587,26.824,154.998
C03200=1061.401,-42.775,-65.158,171.589,26.825,154.998
C03201=1061.407,-42.526,-65.170,171.591,26.827,154.998
C03202=1061.414,-42.276,-65.183,171.592,26.829,154.998
C03203=1061.420,-42.026,-65.196,171.594,26.831,154.998
C03204=1061.425,-41.777,-65.209,171.595,26.833,154.999
C03205=1061.432,-41.528,-65.221,171.597,26.835,154.999
C03206=1061.438,-41.278,-65.234,171.599,26.837,154.999
C03207=1061.444,-41.028,-65.246,171.600,26.839,154.999
C03208=1061.450,-40.779,-65.260,171.602,26.841,154.999
C03209=1061.456,-40.529,-65.272,171.604,26.843,154.999
C03210=1061.463,-40.279,-65.284,171.605,26.845,155.000
C03211=1061.469,-40.030,-65.297,171.607,26.847,155.000
C03212=1061.475,-39.780,-65.310,171.608,26.850,155.000
C03213=1061.481,-39.530,-65.323,171.610,26.851,155.000
C03214=1061.487,-39.281,-65.336,171.612,26.854,155.001
C03215=1061.494,-39.031,-65.348,171.613,26.855,155.001
C03216=1061.500,-38.782,-65.361,171.615,26.858,155.001
C03217=1061.506,-38.532,-65.374,171.616,26.859,155.001
C03218=1061.512,-38.283,-65.387,171.618,26.862,155.001
C03219=1061.518,-38.033,-65.399,171.620,26.864,155.002
C03220=1061.524,-37.783,-65.412,171.621,26.866,155.002
C03221=1061.530,-37.534,-65.425,171.623,26.868,155.002
C03222=1061.536,-37.284,-65.438,171.624,26.870,155.002
C03223=1061.542,-37.035,-65.451,171.626,26.872,155.002
C03224=1061.548,-36.785,-65.464,171.628,26.874,155.003
C03225=1061.554,-36.535,-65.477,171.629,26.876,155.003
C03226=1061.560,-36.286,-65.489,171.631,26.878,155.003
C03227=1061.567,-36.036,-65.503,171.632,26.881,155.003
C03228=1061.573,-35.786,-65.515,171.634,26.882,155.004
C03229=1061.579,-35.537,-65.529,171.636,26.885,155.004
C03230=1061.585,-35.287,-65.541,171.637,26.887,155.004
C03231=1061.591,-35.038,-65.554,171.639,26.889,155.004
C03232=1061.597,-34.789,-65.568,171.640,26.891,155.004
C03233=1061.604,-34.509,-65.582,171.642,26.893,155.005
C03234=1061.610,-34.232,-65.596,171.643,26.895,155.005
C03235=1061.617,-33.953,-65.611,171.646,26.898,155.005
C03236=1061.624,-33.674,-65.626,171.647,26.900,155.006
C03237=1061.630,-33.424,-65.639,171.649,26.903,155.006
C03238=1061.636,-33.175,-65.652,171.651,26.904,155.006
C03239=1061.642,-32.925,-65.665,171.652,26.907,155.006
C03240=1061.648,-32.676,-65.678,171.654,26.909,155.006
C03241=1061.654,-32.426,-65.691,171.655,26.911,155.007
C03242=1061.660,-32.177,-65.704,171.657,26.913,155.007
C03243=1061.667,-31.928,-65.717,171.659,26.915,155.007
C03244=1061.672,-31.678,-65.730,171.660,26.918,155.007
C03245=1061.679,-31.428,-65.743,171.662,26.919,155.008
C03246=1061.686,-31.178,-65.757,171.663,26.922,155.008
C03247=1061.691,-30.928,-65.769,171.665,26.924,155.008
C03248=1061.698,-30.679,-65.782,171.667,26.926,155.008
C03249=1061.704,-30.430,-65.796,171.668,26.928,155.008
C03250=1061.709,-30.180,-65.809,171.670,26.930,155.009
C03251=1061.715,-29.931,-65.822,171.671,26.932,155.009
C03252=1061.721,-29.681,-65.835,171.673,26.934,155.009
C03253=1061.728,-29.431,-65.849,171.675,26.936,155.009
C03254=1061.734,-29.181,-65.862,171.676,26.939,155.010
C03255=1061.740,-28.932,-65.875,171.678,26.941,155.010
C03256=1061.747,-28.683,-65.888,171.679,26.943,155.010
C03257=1061.753,-28.434,-65.901,171.681,26.945,155.010
C03258=1061.759,-28.184,-65.914,171.682,26.947,155.011
C03259=1061.766,-27.934,-65.928,171.684,26.950,155.011
C03260=1061.772,-27.685,-65.941,171.686,26.951,155.011
C03261=1061.777,-27.435,-65.955,171.687,26.954,155.011
C03262=1061.783,-27.185,-65.967,171.689,26.956,155.012
C03263=1061.789,-26.936,-65.981,171.690,26.958,155.012
C03264=1061.796,-26.686,-65.994,171.691,26.960,155.012
C03265=1061.802,-26.437,-66.007,171.693,26.962,155.012
C03266=1061.808,-26.187,-66.021,171.694,26.964,155.013
C03267=1061.814,-25.937,-66.034,171.696,26.967,155.013
C03268=1061.820,-25.688,-66.047,171.697,26.969,155.013
C03269=1061.825,-25.438,-66.061,171.699,26.971,155.013
C03270=1061.832,-25.189,-66.074,171.700,26.973,155.014
C03271=1061.838,-24.939,-66.088,171.702,26.976,155.014
C03272=1061.844,-24.689,-66.102,171.704,26.977,155.014
C03273=1061.850,-24.440,-66.115,171.705,26.980,155.014
C03274=1061.856,-24.190,-66.128,171.707,26.982,155.015
C03275=1061.862,-23.941,-66.141,171.708,26.984,155.015
C03276=1061.868,-23.691,-66.155,171.710,26.987,155.015
C03277=1061.875,-23.441,-66.168,171.712,26.989,155.015
C03278=1061.880,-23.192,-66.182,171.713,26.991,155.016
C03279=1061.886,-22.943,-66.196,171.715,26.993,155.016
C03280=1061.892,-22.693,-66.209,171.716,26.996,155.016
C03281=1061.899,-22.443,-66.223,171.718,26.998,155.016
C03282=1061.905,-22.194,-66.236,171.719,27.000,155.017
C03283=1061.911,-21.945,-66.250,171.721,27.002,155.017
C03284=1061.916,-21.695,-66.263,171.723,27.004,155.017
C03285=1061.923,-21.445,-66.277,171.724,27.007,155.017
C03286=1061.929,-21.196,-66.290,171.726,27.009,155.018
C03287=1061.935,-20.946,-66.304,171.727,27.011,155.018
C03288=1061.941,-20.697,-66.317,171.729,27.013,155.018
C03289=1061.948,-20.447,-66.331,171.730,27.016,155.018
C03290=1061.953,-20.197,-66.345,171.732,27.018,155.019
C03291=1061.960,-19.948,-66.358,171.734,27.020,155.019
C03292=1061.965,-19.699,-66.372,171.735,27.023,155.019
C03293=1061.972,-19.449,-66.386,171.737,27.025,155.020
C03294=1061.978,-19.199,-66.399,171.738,27.027,155.020
C03295=1061.984,-18.950,-66.413,171.740,27.029,155.020
C03296=1061.990,-18.700,-66.427,171.740,27.032,155.020
C03297=1061.997,-18.421,-66.442,171.743,27.034,155.021
C03298=1062.005,-18.142,-66.457,171.745,27.036,155.021
C03299=1062.010,-17.862,-66.472,171.746,27.039,155.021
C03300=1062.018,-17.582,-66.488,171.748,27.042,155.021
C03301=1062.024,-17.333,-66.501,171.749,27.044,155.022
C03302=1062.029,-17.084,-66.515,171.751,27.046,155.022
C03303=1062.037,-16.834,-66.529,171.752,27.048,155.022
C03304=1062.043,-16.585,-66.542,171.754,27.051,155.023
C03305=1062.048,-16.335,-66.556,171.755,27.053,155.023
C03306=1062.055,-16.085,-66.570,171.757,27.055,155.023
C03307=1062.061,-15.836,-66.584,171.759,27.058,155.023
C03308=1062.067,-15.587,-66.597,171.760,27.060,155.024
C03309=1062.073,-15.336,-66.611,171.762,27.062,155.024
C03310=1062.079,-15.088,-66.625,171.763,27.064,155.024
C03311=1062.085,-14.838,-66.639,171.765,27.067,155.024
C03312=1062.092,-14.588,-66.653,171.766,27.069,155.025
C03313=1062.097,-14.339,-66.667,171.768,27.071,155.025
C03314=1062.103,-14.089,-66.680,171.769,27.074,155.025
C03315=1062.110,-13.840,-66.695,171.771,27.076,155.025
C03316=1062.115,-13.590,-66.709,171.773,27.078,155.026
C03317=1062.121,-13.341,-66.722,171.773,27.080,155.026
C03318=1062.127,-13.091,-66.736,171.775,27.082,155.026
C03319=1062.134,-12.842,-66.750,171.776,27.085,155.027
C03320=1062.139,-12.592,-66.764,171.778,27.088,155.027
C03321=1062.146,-12.342,-66.778,171.779,27.090,155.027
C03322=1062.152,-12.093,-66.792,171.781,27.092,155.028
C03323=1062.158,-11.844,-66.806,171.783,27.094,155.028
C03324=1062.164,-11.594,-66.820,171.784,27.097,155.028
C03325=1062.170,-11.344,-66.834,171.786,27.099,155.028
C03326=1062.176,-11.094,-66.848,171.787,27.101,155.029
C03327=1062.182,-10.845,-66.862,171.789,27.104,155.029
C03328=1062.188,-10.596,-66.876,171.790,27.106,155.029
C03329=1062.194,-10.346,-66.890,171.792,27.109,155.030
C03330=1062.201,-10.097,-66.904,171.793,27.111,155.030
C03331=1062.206,-9.847,-66.918,171.795,27.113,155.030
C03332=1062.212,-9.597,-66.932,171.797,27.116,155.030
C03333=1062.219,-9.348,-66.946,171.798,27.118,155.031
C03334=1062.225,-9.098,-66.960,171.800,27.120,155.031
C03335=1062.230,-8.849,-66.975,171.800,27.122,155.031
C03336=1062.237,-8.599,-66.988,171.802,27.125,155.032
C03337=1062.243,-8.350,-67.002,171.803,27.127,155.032
C03338=1062.249,-8.101,-67.017,171.805,27.130,155.032
C03339=1062.255,-7.851,-67.030,171.807,27.132,155.032
C03340=1062.261,-7.602,-67.045,171.808,27.134,155.033
C03341=1062.267,-7.351,-67.059,171.810,27.136,155.033
C03342=1062.273,-7.102,-67.073,171.811,27.139,155.033
C03343=1062.280,-6.853,-67.088,171.813,27.141,155.034
C03344=1062.285,-6.603,-67.101,171.814,27.144,155.034
C03345=1062.292,-6.354,-67.116,171.816,27.146,155.034
C03346=1062.298,-6.104,-67.130,171.818,27.148,155.034
C03347=1062.304,-5.855,-67.144,171.819,27.151,155.035
C03348=1062.310,-5.605,-67.158,171.821,27.153,155.035
C03349=1062.316,-5.356,-67.172,171.822,27.155,155.035
C03350=1062.322,-5.106,-67.187,171.824,27.158,155.036
C03351=1062.328,-4.857,-67.201,171.824,27.160,155.036
C03352=1062.335,-4.607,-67.215,171.826,27.162,155.036
C03353=1062.341,-4.358,-67.229,171.828,27.165,155.036
C03354=1062.347,-4.108,-67.244,171.829,27.167,155.037
C03355=1062.353,-3.859,-67.258,171.831,27.169,155.037
C03356=1062.359,-3.609,-67.272,171.832,27.171,155.037
C03357=1062.366,-3.359,-67.287,171.834,27.174,155.038
C03358=1062.371,-3.110,-67.301,171.835,27.177,155.038
C03359=1062.377,-2.861,-67.315,171.837,27.179,155.038
C03360=1062.383,-2.610,-67.329,171.838,27.182,155.039
C03361=1062.390,-2.330,-67.346,171.840,27.184,155.039
C03362=1062.397,-2.049,-67.362,171.841,27.187,155.039
C03363=1062.404,-1.768,-67.379,171.843,27.190,155.040
C03364=1062.411,-1.487,-67.394,171.844,27.193,155.040
C03365=1062.416,-1.238,-67.409,171.846,27.195,155.040
C03366=1062.422,-0.988,-67.423,171.848,27.197,155.040
C03367=1062.428,-0.739,-67.438,171.849,27.200,155.041
C03368=1062.434,-0.490,-67.452,171.851,27.202,155.041
C03369=1062.440,-0.239,-67.467,171.852,27.205,155.041
C03370=1062.446,0.010,-67.481,171.854,27.207,155.042
C03371=1062.452,0.259,-67.496,171.855,27.210,155.042
C03372=1062.458,0.509,-67.510,171.857,27.212,155.042
C03373=1062.464,0.729,-67.523,171.858,27.214,155.043
C03374=1062.469,0.949,-67.537,171.859,27.216,155.043
C03375=1062.474,1.169,-67.549,171.861,27.218,155.043
C03376=1062.479,1.390,-67.562,171.862,27.221,155.043
C03377=1062.485,1.609,-67.575,171.863,27.223,155.044
C03378=1062.489,1.830,-67.588,171.864,27.225,155.044
C03379=1062.495,2.050,-67.600,171.866,27.227,155.044
C03380=1062.501,2.270,-67.613,171.867,27.229,155.045
C03381=1062.507,2.520,-67.628,171.868,27.232,155.045
C03382=1062.512,2.769,-67.642,171.870,27.234,155.045
C03383=1062.519,3.019,-67.657,171.871,27.237,155.046
C03384=1062.525,3.268,-67.672,171.873,27.239,155.046
C03385=1062.531,3.517,-67.687,171.874,27.242,155.046
C03386=1062.536,3.767,-67.701,171.876,27.244,155.046
C03387=1062.543,4.017,-67.716,171.877,27.246,155.047
C03388=1062.549,4.266,-67.730,171.879,27.249,155.047
C03389=1062.555,4.515,-67.745,171.881,27.252,155.047
C03390=1062.561,4.765,-67.760,171.881,27.254,155.048
C03391=1062.567,5.014,-67.774,171.883,27.256,155.048
C03392=1062.573,5.264,-67.789,171.884,27.259,155.048
C03393=1062.580,5.514,-67.804,171.886,27.261,155.049
C03394=1062.585,5.763,-67.818,171.887,27.264,155.049
C03395=1062.591,6.013,-67.834,171.889,27.266,155.049
C03396=1062.597,6.262,-67.848,171.890,27.268,155.050
C03397=1062.603,6.512,-67.863,171.892,27.271,155.050
C03398=1062.609,6.762,-67.878,171.894,27.273,155.050
C03399=1062.615,7.011,-67.892,171.895,27.276,155.051
C03400=1062.621,7.260,-67.907,171.897,27.279,155.051
C03401=1062.628,7.510,-67.922,171.898,27.281,155.051
C03402=1062.634,7.759,-67.937,171.899,27.283,155.052
C03403=1062.640,8.008,-67.952,171.900,27.286,155.052
C03404=1062.646,8.257,-67.966,171.902,27.288,155.052
C03405=1062.652,8.507,-67.981,171.903,27.291,155.053
C03406=1062.659,8.757,-67.996,171.905,27.293,155.053
C03407=1062.664,9.006,-68.011,171.907,27.295,155.053
C03408=1062.670,9.256,-68.025,171.908,27.298,155.053
C03409=1062.677,9.506,-68.040,171.910,27.300,155.054
C03410=1062.682,9.756,-68.055,171.911,27.303,155.054
C03411=1062.688,10.005,-68.070,171.913,27.306,155.054
C03412=1062.695,10.254,-68.085,171.914,27.308,155.055
C03413=1062.701,10.504,-68.100,171.915,27.310,155.055
C03414=1062.707,10.753,-68.114,171.916,27.313,155.055
C03415=1062.713,11.002,-68.129,171.918,27.315,155.056
C03416=1062.719,11.252,-68.144,171.919,27.318,155.056
C03417=1062.725,11.501,-68.159,171.921,27.320,155.056
C03418=1062.732,11.751,-68.174,171.923,27.322,155.057
C03419=1062.738,12.000,-68.189,171.924,27.325,155.057
C03420=1062.744,12.250,-68.204,171.926,27.327,155.057
C03421=1062.749,12.499,-68.219,171.927,27.330,155.058
C03422=1062.756,12.748,-68.235,171.929,27.333,155.058
C03423=1062.763,12.998,-68.250,171.929,27.335,155.058
C03424=1062.769,13.248,-68.264,171.931,27.337,155.059
C03425=1062.777,13.589,-68.285,171.933,27.341,155.059
C03426=1062.785,13.931,-68.306,171.936,27.344,155.059
C03427=1062.795,14.272,-68.326,171.937,27.347,155.060
C03428=1062.802,14.613,-68.346,171.940,27.351,155.060
C03429=1062.808,14.863,-68.362,171.941,27.354,155.061
C03430=1062.814,15.113,-68.377,171.943,27.356,155.061
C03431=1062.820,15.362,-68.391,171.943,27.358,155.061
C03432=1062.826,15.612,-68.407,171.945,27.361,155.062
C03433=1062.832,15.861,-68.422,171.946,27.364,155.062
C03434=1062.839,16.110,-68.438,171.948,27.366,155.062
C03435=1062.844,16.360,-68.453,171.949,27.369,155.063
C03436=1062.850,16.609,-68.468,171.951,27.371,155.063
C03437=1062.857,16.859,-68.483,171.952,27.374,155.063
C03438=1062.862,17.109,-68.498,171.954,27.376,155.064
C03439=1062.868,17.358,-68.513,171.956,27.379,155.064
C03440=1062.875,17.607,-68.528,171.957,27.381,155.064
C03441=1062.881,17.857,-68.544,171.958,27.384,155.065
C03442=1062.887,18.107,-68.559,171.959,27.386,155.065
C03443=1062.892,18.356,-68.574,171.961,27.389,155.065
C03444=1062.899,18.605,-68.590,171.962,27.391,155.066
C03445=1062.905,18.855,-68.605,171.964,27.394,155.066
C03446=1062.911,19.105,-68.620,171.965,27.396,155.066
C03447=1062.917,19.354,-68.635,171.967,27.399,155.067
C03448=1062.923,19.603,-68.650,171.969,27.401,155.067
C03449=1062.929,19.853,-68.666,171.970,27.404,155.067
C03450=1062.935,20.102,-68.681,171.971,27.406,155.068
C03451=1062.941,20.352,-68.697,171.972,27.409,155.068
C03452=1062.948,20.601,-68.712,171.974,27.411,155.068
C03453=1062.953,20.850,-68.727,171.975,27.414,155.069
C03454=1062.959,21.099,-68.743,171.977,27.416,155.069
C03455=1062.966,21.349,-68.758,171.978,27.419,155.069
C03456=1062.971,21.599,-68.773,171.980,27.421,155.070
C03457=1062.978,21.848,-68.789,171.981,27.424,155.070
C03458=1062.983,22.097,-68.804,171.983,27.427,155.070
C03459=1062.989,22.347,-68.819,171.984,27.429,155.071
C03460=1062.995,22.596,-68.835,171.985,27.432,155.071
C03461=1063.002,22.846,-68.850,171.987,27.434,155.071
C03462=1063.007,23.096,-68.866,171.988,27.437,155.072
C03463=1063.013,23.344,-68.881,171.990,27.439,155.072
C03464=1063.019,23.594,-68.897,171.991,27.442,155.072
C03465=1063.026,23.843,-68.912,171.993,27.444,155.073
C03466=1063.031,24.093,-68.928,171.994,27.447,155.073
C03467=1063.038,24.342,-68.944,171.996,27.450,155.073
C03468=1063.044,24.592,-68.959,171.997,27.452,155.074
C03469=1063.050,24.842,-68.974,171.998,27.455,155.074
C03470=1063.056,25.091,-68.990,172.000,27.457,155.074
C03471=1063.062,25.340,-69.005,172.001,27.460,155.075
C03472=1063.068,25.590,-69.021,172.003,27.462,155.075
C03473=1063.074,25.840,-69.037,172.004,27.465,155.075
C03474=1063.080,26.089,-69.052,172.006,27.467,155.076
C03475=1063.086,26.339,-69.068,172.007,27.470,155.076
C03476=1063.093,26.588,-69.084,172.009,27.473,155.077
C03477=1063.098,26.838,-69.099,172.009,27.475,155.077
C03478=1063.105,27.087,-69.115,172.011,27.478,155.077
C03479=1063.110,27.336,-69.130,172.013,27.480,155.078
C03480=1063.117,27.585,-69.146,172.014,27.483,155.078
C03481=1063.122,27.835,-69.161,172.016,27.485,155.078
C03482=1063.128,28.084,-69.177,172.017,27.488,155.079
C03483=1063.135,28.333,-69.193,172.019,27.491,155.079
C03484=1063.141,28.583,-69.209,172.020,27.493,155.079
C03485=1063.147,28.832,-69.224,172.021,27.496,155.080
C03486=1063.153,29.082,-69.240,172.022,27.498,155.080
C03487=1063.159,29.332,-69.256,172.024,27.501,155.080
C03488=1063.164,29.582,-69.272,172.025,27.504,155.081
C03489=1063.172,29.866,-69.290,172.027,27.506,155.081
C03490=1063.178,30.149,-69.307,172.028,27.509,155.082
C03491=1063.185,30.434,-69.325,172.031,27.512,155.082
C03492=1063.192,30.717,-69.343,172.032,27.515,155.082
C03493=1063.198,30.967,-69.360,172.034,27.518,155.083
C03494=1063.203,31.217,-69.375,172.034,27.521,155.083
C03495=1063.210,31.466,-69.391,172.036,27.523,155.083
C03496=1063.216,31.715,-69.407,172.038,27.526,155.084
C03497=1063.222,31.965,-69.423,172.039,27.528,155.084
C03498=1063.228,32.214,-69.439,172.041,27.531,155.084
C03499=1063.234,32.463,-69.454,172.042,27.534,155.085
C03500=1063.240,32.713,-69.470,172.044,27.536,155.085
C03501=1063.246,32.963,-69.486,172.045,27.539,155.085
C03502=1063.252,33.212,-69.503,172.046,27.541,155.086
C03503=1063.259,33.461,-69.518,172.047,27.544,155.086
C03504=1063.264,33.711,-69.534,172.049,27.546,155.087
C03505=1063.270,33.960,-69.550,172.050,27.549,155.087
C03506=1063.276,34.210,-69.566,172.052,27.552,155.087
C03507=1063.283,34.459,-69.582,172.054,27.554,155.088
C03508=1063.288,34.709,-69.597,172.055,27.557,155.088
C03509=1063.294,34.958,-69.614,172.057,27.559,155.088
C03510=1063.300,35.208,-69.630,172.057,27.562,155.089
C03511=1063.306,35.457,-69.646,172.059,27.565,155.089
C03512=1063.313,35.707,-69.661,172.060,27.567,155.089
C03513=1063.319,35.956,-69.677,172.062,27.570,155.090
C03514=1063.325,36.205,-69.694,172.063,27.573,155.090
C03515=1063.331,36.455,-69.710,172.065,27.575,155.090
C03516=1063.337,36.704,-69.726,172.067,27.578,155.091
C03517=1063.343,36.953,-69.742,172.068,27.580,155.091
C03518=1063.349,37.203,-69.757,172.070,27.583,155.092
C03519=1063.355,37.452,-69.774,172.070,27.585,155.092
C03520=1063.361,37.702,-69.790,172.072,27.588,155.092
C03521=1063.367,37.951,-69.806,172.073,27.590,155.093
C03522=1063.373,38.200,-69.822,172.075,27.593,155.093
C03523=1063.379,38.449,-69.838,172.076,27.596,155.093
C03524=1063.385,38.699,-69.854,172.078,27.598,155.094
C03525=1063.391,38.948,-69.871,172.079,27.601,155.094
C03526=1063.397,39.198,-69.886,172.081,27.604,155.094
C03527=1063.403,39.447,-69.902,172.082,27.606,155.095
C03528=1063.409,39.697,-69.919,172.083,27.609,155.095
C03529=1063.415,39.946,-69.935,172.085,27.612,155.096
C03530=1063.421,40.195,-69.951,172.086,27.614,155.096
C03531=1063.427,40.445,-69.967,172.088,27.617,155.096
C03532=1063.433,40.694,-69.984,172.089,27.619,155.097
C03533=1063.439,40.943,-70.000,172.091,27.622,155.097
C03534=1063.444,41.193,-70.016,172.092,27.625,155.097
C03535=1063.450,41.442,-70.032,172.093,27.627,155.098
C03536=1063.456,41.691,-70.049,172.095,27.630,155.098
C03537=1063.462,41.941,-70.065,172.096,27.633,155.098
C03538=1063.469,42.191,-70.082,172.098,27.636,155.099
C03539=1063.475,42.440,-70.098,172.099,27.638,155.099
C03540=1063.481,42.690,-70.114,172.101,27.641,155.100
C03541=1063.487,42.939,-70.130,172.102,27.643,155.100
C03542=1063.493,43.188,-70.147,172.104,27.646,155.100
C03543=1063.499,43.438,-70.163,172.104,27.648,155.101
C03544=1063.505,43.687,-70.179,172.106,27.651,155.101
C03545=1063.510,43.937,-70.196,172.107,27.654,155.101
C03546=1063.516,44.186,-70.212,172.109,27.657,155.102
C03547=1063.522,44.435,-70.228,172.111,27.659,155.102
C03548=1063.528,44.684,-70.245,172.112,27.662,155.103
C03549=1063.534,44.933,-70.262,172.114,27.665,155.103
C03550=1063.539,45.183,-70.279,172.114,27.667,155.103
C03551=1063.545,45.432,-70.295,172.116,27.670,155.104
C03552=1063.552,45.682,-70.311,172.117,27.673,155.104
C03553=1063.558,45.967,-70.330,172.119,27.676,155.105
C03554=1063.565,46.251,-70.349,172.120,27.678,155.105
C03555=1063.571,46.534,-70.368,172.123,27.682,155.105
C03556=1063.578,46.819,-70.387,172.124,27.685,155.106
C03557=1063.584,47.068,-70.403,172.126,27.688,155.106
C03558=1063.590,47.317,-70.419,172.126,27.690,155.107
C03559=1063.595,47.566,-70.437,172.128,27.693,155.107
C03560=1063.602,47.816,-70.453,172.129,27.695,155.107
C03561=1063.608,48.066,-70.470,172.131,27.698,155.108
C03562=1063.614,48.315,-70.486,172.132,27.701,155.108
C03563=1063.619,48.565,-70.503,172.134,27.704,155.108
C03564=1063.625,48.813,-70.520,172.135,27.707,155.109
C03565=1063.631,49.063,-70.536,172.137,27.709,155.109
C03566=1063.637,49.312,-70.552,172.138,27.711,155.110
C03567=1063.642,49.562,-70.569,172.139,27.714,155.110
C03568=1063.649,49.811,-70.586,172.141,27.717,155.110
C03569=1063.655,50.061,-70.603,172.142,27.720,155.111
C03570=1063.660,50.310,-70.619,172.144,27.722,155.111
C03571=1063.666,50.560,-70.636,172.145,27.725,155.111
C03572=1063.673,50.808,-70.653,172.147,27.728,155.112
C03573=1063.679,51.058,-70.669,172.148,27.731,155.112
C03574=1063.684,51.308,-70.686,172.149,27.733,155.113
C03575=1063.691,51.557,-70.703,172.150,27.736,155.113
C03576=1063.697,51.806,-70.719,172.152,27.738,155.113
C03577=1063.703,52.056,-70.736,172.154,27.741,155.114
C03578=1063.708,52.305,-70.753,172.155,27.744,155.114
C03579=1063.715,52.555,-70.770,172.157,27.747,155.114
C03580=1063.721,52.804,-70.786,172.158,27.749,155.115
C03581=1063.726,53.053,-70.804,172.160,27.752,155.115
C03582=1063.732,53.302,-70.820,172.160,27.754,155.116
C03583=1063.738,53.552,-70.836,172.162,27.757,155.116
C03584=1063.744,53.801,-70.854,172.163,27.760,155.116
C03585=1063.750,54.051,-70.870,172.165,27.762,155.117
C03586=1063.756,54.299,-70.887,172.167,27.765,155.117
C03587=1063.762,54.549,-70.904,172.168,27.768,155.117
C03588=1063.768,54.799,-70.921,172.170,27.770,155.118
C03589=1063.774,55.048,-70.938,172.171,27.773,155.118
C03590=1063.780,55.297,-70.954,172.172,27.775,155.119
C03591=1063.786,55.546,-70.972,172.173,27.778,155.119
C03592=1063.792,55.796,-70.988,172.175,27.781,155.119
C03593=1063.799,56.045,-71.005,172.176,27.784,155.120
C03594=1063.804,56.295,-71.022,172.178,27.786,155.120
C03595=1063.810,56.544,-71.038,172.180,27.789,155.120
C03596=1063.817,56.794,-71.056,172.181,27.792,155.121
C03597=1063.822,57.043,-71.073,172.183,27.794,155.121
C03598=1063.828,57.292,-71.089,172.183,27.797,155.122
C03599=1063.835,57.542,-71.106,172.185,27.799,155.122
C03600=1063.840,57.791,-71.124,172.186,27.802,155.122
C03601=1063.846,58.040,-71.140,172.188,27.805,155.123
C03602=1063.852,58.289,-71.157,172.189,27.808,155.123
C03603=1063.859,58.539,-71.175,172.191,27.810,155.123
C03604=1063.864,58.788,-71.191,172.193,27.813,155.124
C03605=1063.870,59.037,-71.209,172.194,27.815,155.124
C03606=1063.877,59.287,-71.225,172.195,27.818,155.125
C03607=1063.883,59.536,-71.242,172.196,27.820,155.125
C03608=1063.888,59.786,-71.259,172.198,27.823,155.125
C03609=1063.895,60.035,-71.276,172.199,27.826,155.126
C03610=1063.901,60.284,-71.293,172.201,27.829,155.126
C03611=1063.906,60.533,-71.310,172.203,27.831,155.126
C03612=1063.913,60.783,-71.328,172.204,27.834,155.127
C03613=1063.919,61.032,-71.344,172.206,27.836,155.127
C03614=1063.925,61.282,-71.362,172.207,27.839,155.128
C03615=1063.931,61.531,-71.378,172.208,27.841,155.128
C03616=1063.937,61.780,-71.396,172.209,27.844,155.128
C03617=1063.944,62.065,-71.415,172.211,27.847,155.129
C03618=1063.951,62.348,-71.435,172.213,27.850,155.129
C03619=1063.958,62.632,-71.454,172.215,27.853,155.129
C03620=1063.965,62.916,-71.474,172.216,27.856,155.130
C03621=1063.971,63.165,-71.491,172.218,27.859,155.130
C03622=1063.977,63.415,-71.508,172.220,27.861,155.131
